C03642=1066.521,27.766,432.620,172.399,26.126,154.782
C03643=1066.516,27.517,432.635,172.398,26.123,154.782
C03644=1066.510,27.267,432.651,172.397,26.120,154.781
C03645=1066.504,27.017,432.666,172.395,26.118,154.781
C03646=1066.497,26.768,432.682,172.394,26.115,154.780
C03647=1066.492,26.518,432.698,172.392,26.112,154.780
C03648=1066.485,26.269,432.713,172.391,26.109,154.780
C03649=1066.480,26.020,432.728,172.389,26.107,154.780
C03650=1066.473,25.771,432.743,172.388,26.104,154.779
C03651=1066.467,25.521,432.760,172.386,26.102,154.779
C03652=1066.461,25.272,432.775,172.385,26.099,154.778
C03653=1066.455,25.022,432.790,172.384,26.096,154.778
C03654=1066.449,24.773,432.805,172.382,26.094,154.778
C03655=1066.444,24.523,432.821,172.381,26.091,154.777
C03656=1066.437,24.274,432.836,172.379,26.089,154.777
C03657=1066.431,24.024,432.852,172.378,26.086,154.777
C03658=1066.425,23.775,432.867,172.376,26.084,154.776
C03659=1066.420,23.525,432.882,172.375,26.081,154.776
C03660=1066.413,23.276,432.898,172.374,26.078,154.776
C03661=1066.408,23.026,432.913,172.372,26.075,154.775
C03662=1066.401,22.777,432.928,172.371,26.073,154.775
C03663=1066.396,22.527,432.944,172.369,26.070,154.775
C03664=1066.389,22.278,432.959,172.368,26.068,154.774
C03665=1066.384,22.028,432.975,172.366,26.065,154.774
C03666=1066.377,21.779,432.990,172.366,26.062,154.774
C03667=1066.372,21.529,433.005,172.365,26.060,154.773
C03668=1066.366,21.280,433.021,172.363,26.057,154.773
C03669=1066.360,21.030,433.036,172.362,26.055,154.773
C03670=1066.354,20.781,433.051,172.360,26.052,154.772
C03671=1066.348,20.532,433.066,172.359,26.050,154.772
C03672=1066.342,20.283,433.082,172.357,26.047,154.772
C03673=1066.336,20.033,433.097,172.356,26.045,154.771
C03674=1066.330,19.783,433.112,172.355,26.042,154.771
C03675=1066.324,19.534,433.127,172.353,26.039,154.771
C03676=1066.318,19.284,433.142,172.352,26.037,154.770
C03677=1066.312,19.034,433.157,172.350,26.034,154.770
C03678=1066.305,18.785,433.173,172.349,26.031,154.770
C03679=1066.300,18.536,433.188,172.347,26.029,154.769
C03680=1066.294,18.286,433.203,172.346,26.026,154.769
C03681=1066.288,18.037,433.218,172.344,26.024,154.769
C03682=1066.282,17.788,433.233,172.343,26.021,154.768
C03683=1066.276,17.538,433.248,172.342,26.019,154.768
C03684=1066.270,17.288,433.263,172.340,26.016,154.768
C03685=1066.264,17.040,433.279,172.339,26.013,154.767
C03686=1066.258,16.790,433.294,172.337,26.011,154.767
C03687=1066.252,16.540,433.309,172.336,26.008,154.767
C03688=1066.246,16.291,433.324,172.335,26.005,154.766
C03689=1066.240,16.041,433.339,172.333,26.003,154.766
C03690=1066.234,15.792,433.354,172.332,26.000,154.766
C03691=1066.228,15.543,433.369,172.330,25.998,154.765
C03692=1066.222,15.293,433.384,172.329,25.995,154.765
C03693=1066.216,15.043,433.399,172.327,25.993,154.765
C03694=1066.210,14.794,433.414,172.326,25.990,154.764
C03695=1066.203,14.511,433.431,172.324,25.987,154.764
C03696=1066.196,14.230,433.448,172.323,25.984,154.764
C03697=1066.189,13.948,433.465,172.322,25.982,154.763
C03698=1066.182,13.665,433.482,172.320,25.979,154.763
C03699=1066.176,13.416,433.497,172.319,25.976,154.763
C03700=1066.170,13.167,433.511,172.317,25.974,154.762
C03701=1066.164,12.917,433.527,172.316,25.971,154.762
C03702=1066.158,12.667,433.542,172.314,25.969,154.762
C03703=1066.152,12.418,433.556,172.313,25.966,154.761
C03704=1066.146,12.169,433.571,172.312,25.964,154.761
C03705=1066.140,11.919,433.586,172.310,25.961,154.761
C03706=1066.134,11.670,433.601,172.309,25.958,154.760
C03707=1066.128,11.420,433.615,172.307,25.956,154.760
C03708=1066.121,11.170,433.630,172.306,25.953,154.760
C03709=1066.115,10.921,433.644,172.304,25.951,154.759
C03710=1066.109,10.671,433.659,172.303,25.949,154.759
C03711=1066.103,10.422,433.674,172.302,25.946,154.759
C03712=1066.098,10.172,433.690,172.300,25.943,154.758
C03713=1066.091,9.923,433.704,172.299,25.941,154.758
C03714=1066.086,9.674,433.719,172.297,25.938,154.758
C03715=1066.079,9.424,433.734,172.296,25.936,154.757
C03716=1066.073,9.174,433.748,172.294,25.934,154.757
C03717=1066.067,8.925,433.763,172.293,25.931,154.757
C03718=1066.061,8.675,433.778,172.291,25.928,154.757
C03719=1066.055,8.426,433.792,172.290,25.925,154.756
C03720=1066.049,8.177,433.807,172.289,25.923,154.756
C03721=1066.042,7.927,433.822,172.287,25.921,154.756
C03722=1066.037,7.677,433.836,172.286,25.918,154.755
C03723=1066.030,7.428,433.851,172.284,25.916,154.755
C03724=1066.025,7.179,433.866,172.283,25.913,154.755
C03725=1066.018,6.929,433.881,172.281,25.910,154.754
C03726=1066.012,6.680,433.895,172.280,25.908,154.754
C03727=1066.006,6.430,433.909,172.278,25.906,154.754
C03728=1066.000,6.180,433.924,172.277,25.903,154.753
C03729=1065.994,5.931,433.939,172.276,25.901,154.753
C03730=1065.988,5.682,433.954,172.274,25.898,154.753
C03731=1065.982,5.432,433.968,172.273,25.895,154.752
C03732=1065.976,5.182,433.983,172.271,25.893,154.752
C03733=1065.970,4.934,433.997,172.270,25.890,154.752
C03734=1065.964,4.684,434.012,172.268,25.888,154.751
C03735=1065.958,4.434,434.026,172.267,25.885,154.751
C03736=1065.952,4.185,434.041,172.266,25.883,154.751
C03737=1065.946,3.936,434.056,172.265,25.881,154.751
C03738=1065.940,3.685,434.070,172.264,25.878,154.750
C03739=1065.934,3.436,434.084,172.262,25.875,154.750
C03740=1065.928,3.187,434.099,172.261,25.873,154.750
C03741=1065.923,2.937,434.113,172.259,25.871,154.749
C03742=1065.916,2.688,434.128,172.258,25.868,154.749
C03743=1065.910,2.439,434.143,172.256,25.865,154.749
C03744=1065.904,2.188,434.157,172.255,25.863,154.748
C03745=1065.898,1.939,434.172,172.254,25.860,154.748
C03746=1065.892,1.690,434.186,172.252,25.858,154.748
C03747=1065.887,1.440,434.200,172.251,25.856,154.747
C03748=1065.880,1.190,434.215,172.249,25.853,154.747
C03749=1065.875,0.941,434.229,172.248,25.850,154.747
C03750=1065.868,0.691,434.244,172.246,25.848,154.746
C03751=1065.863,0.442,434.259,172.245,25.845,154.746
C03752=1065.857,0.192,434.273,172.243,25.843,154.746
C03753=1065.851,-0.057,434.287,172.242,25.840,154.746
C03754=1065.845,-0.307,434.301,172.241,25.838,154.745
C03755=1065.839,-0.556,434.316,172.239,25.835,154.745
C03756=1065.833,-0.806,434.330,172.238,25.833,154.745
C03757=1065.827,-1.055,434.345,172.236,25.830,154.744
C03758=1065.822,-1.305,434.359,172.235,25.828,154.744
C03759=1065.815,-1.585,434.375,172.233,25.825,154.744
C03760=1065.808,-1.865,434.391,172.232,25.822,154.743
C03761=1065.801,-2.145,434.408,172.230,25.819,154.743
C03762=1065.794,-2.425,434.424,172.228,25.816,154.743
C03763=1065.788,-2.675,434.438,172.227,25.814,154.742
C03764=1065.783,-2.924,434.452,172.225,25.811,154.742
C03765=1065.777,-3.174,434.466,172.224,25.809,154.742
C03766=1065.771,-3.424,434.481,172.223,25.806,154.741
C03767=1065.765,-3.673,434.495,172.221,25.804,154.741
C03768=1065.758,-3.923,434.509,172.220,25.801,154.741
C03769=1065.753,-4.172,434.523,172.218,25.799,154.740
C03770=1065.747,-4.422,434.538,172.217,25.797,154.740
C03771=1065.740,-4.671,434.552,172.215,25.794,154.740
C03772=1065.734,-4.921,434.566,172.214,25.792,154.740
C03773=1065.728,-5.171,434.580,172.212,25.789,154.739
C03774=1065.722,-5.419,434.594,172.211,25.787,154.739
C03775=1065.716,-5.669,434.608,172.209,25.784,154.739
C03776=1065.710,-5.918,434.622,172.208,25.782,154.738
C03777=1065.704,-6.169,434.637,172.207,25.780,154.738
C03778=1065.698,-6.418,434.650,172.205,25.777,154.738
C03779=1065.691,-6.668,434.665,172.204,25.775,154.738
C03780=1065.686,-6.917,434.679,172.202,25.772,154.737
C03781=1065.680,-7.166,434.692,172.201,25.770,154.737
C03782=1065.673,-7.416,434.707,172.199,25.767,154.737
C03783=1065.667,-7.665,434.720,172.198,25.765,154.736
C03784=1065.661,-7.916,434.735,172.196,25.763,154.736
C03785=1065.655,-8.165,434.749,172.195,25.760,154.736
C03786=1065.649,-8.414,434.762,172.193,25.758,154.735
C03787=1065.643,-8.664,434.777,172.192,25.755,154.735
C03788=1065.637,-8.913,434.791,172.191,25.753,154.735
C03789=1065.631,-9.162,434.804,172.189,25.751,154.735
C03790=1065.625,-9.413,434.819,172.188,25.748,154.734
C03791=1065.619,-9.662,434.833,172.186,25.746,154.734
C03792=1065.613,-9.911,434.847,172.185,25.743,154.734
C03793=1065.607,-10.161,434.861,172.183,25.741,154.733
C03794=1065.601,-10.410,434.874,172.182,25.738,154.733
C03795=1065.595,-10.660,434.888,172.180,25.736,154.733
C03796=1065.589,-10.910,434.903,172.179,25.734,154.733
C03797=1065.583,-11.159,434.916,172.177,25.731,154.732
C03798=1065.577,-11.408,434.930,172.176,25.729,154.732
C03799=1065.571,-11.659,434.944,172.174,25.727,154.732
C03800=1065.565,-11.908,434.957,172.173,25.724,154.731
C03801=1065.559,-12.157,434.972,172.172,25.721,154.731
C03802=1065.552,-12.407,434.986,172.170,25.719,154.731
C03803=1065.547,-12.657,435.000,172.169,25.717,154.731
C03804=1065.541,-12.906,435.013,172.167,25.714,154.730
C03805=1065.535,-13.155,435.027,172.166,25.712,154.730
C03806=1065.529,-13.406,435.041,172.164,25.710,154.730
C03807=1065.522,-13.654,435.055,172.163,25.707,154.730
C03808=1065.517,-13.904,435.069,172.161,25.704,154.729
C03809=1065.511,-14.153,435.083,172.160,25.702,154.729
C03810=1065.505,-14.403,435.096,172.159,25.700,154.729
C03811=1065.499,-14.653,435.110,172.157,25.697,154.728
C03812=1065.493,-14.902,435.123,172.156,25.695,154.728
C03813=1065.487,-15.153,435.138,172.154,25.693,154.728
C03814=1065.481,-15.402,435.151,172.153,25.690,154.728
C03815=1065.475,-15.651,435.165,172.151,25.688,154.727
C03816=1065.469,-15.901,435.178,172.150,25.686,154.727
C03817=1065.462,-16.150,435.192,172.148,25.683,154.727
C03818=1065.456,-16.400,435.206,172.147,25.681,154.726
C03819=1065.450,-16.649,435.220,172.145,25.679,154.726
C03820=1065.444,-16.899,435.234,172.144,25.676,154.726
C03821=1065.438,-17.148,435.247,172.142,25.674,154.726
C03822=1065.432,-17.398,435.260,172.141,25.672,154.725
C03823=1065.425,-17.676,435.275,172.139,25.669,154.725
C03824=1065.418,-17.955,435.291,172.138,25.666,154.725
C03825=1065.411,-18.234,435.306,172.137,25.664,154.724
C03826=1065.405,-18.513,435.321,172.134,25.661,154.724
C03827=1065.398,-18.762,435.334,172.133,25.659,154.724
C03828=1065.393,-19.011,435.348,172.131,25.657,154.724
C03829=1065.387,-19.261,435.361,172.130,25.654,154.723
C03830=1065.380,-19.511,435.375,172.128,25.652,154.723
C03831=1065.374,-19.760,435.389,172.127,25.650,154.723
C03832=1065.368,-20.009,435.402,172.125,25.647,154.723
C03833=1065.363,-20.259,435.416,172.124,25.645,154.722
C03834=1065.356,-20.509,435.429,172.122,25.643,154.722
C03835=1065.350,-20.758,435.443,172.121,25.640,154.722
C03836=1065.344,-21.008,435.457,172.120,25.638,154.722
C03837=1065.338,-21.257,435.470,172.118,25.636,154.721
C03838=1065.332,-21.506,435.483,172.117,25.633,154.721
C03839=1065.326,-21.757,435.497,172.115,25.631,154.721
C03840=1065.320,-22.007,435.510,172.114,25.629,154.720
C03841=1065.314,-22.256,435.523,172.112,25.626,154.720
C03842=1065.308,-22.505,435.537,172.111,25.625,154.720
C03843=1065.302,-22.755,435.550,172.109,25.622,154.720
C03844=1065.296,-23.004,435.564,172.108,25.620,154.720
C03845=1065.290,-23.254,435.578,172.106,25.618,154.719
C03846=1065.284,-23.504,435.590,172.105,25.615,154.719
C03847=1065.277,-23.753,435.604,172.103,25.613,154.719
C03848=1065.271,-24.003,435.617,172.102,25.610,154.718
C03849=1065.266,-24.252,435.631,172.100,25.608,154.718
C03850=1065.260,-24.501,435.644,172.099,25.606,154.718
C03851=1065.253,-24.751,435.657,172.097,25.603,154.718
C03852=1065.248,-25.002,435.671,172.096,25.601,154.717
C03853=1065.241,-25.251,435.684,172.095,25.599,154.717
C03854=1065.235,-25.500,435.697,172.093,25.596,154.717
C03855=1065.230,-25.750,435.711,172.091,25.595,154.717
C03856=1065.224,-26.000,435.724,172.090,25.592,154.716
C03857=1065.218,-26.249,435.737,172.089,25.590,154.716
C03858=1065.211,-26.498,435.750,172.087,25.588,154.716
C03859=1065.206,-26.748,435.764,172.086,25.585,154.716
C03860=1065.200,-26.998,435.777,172.084,25.583,154.715
C03861=1065.193,-27.248,435.790,172.083,25.581,154.715
C03862=1065.187,-27.497,435.804,172.081,25.579,154.715
C03863=1065.181,-27.747,435.816,172.080,25.576,154.715
C03864=1065.175,-27.996,435.829,172.078,25.574,154.714
C03865=1065.169,-28.245,435.843,172.077,25.572,154.714
C03866=1065.162,-28.494,435.856,172.075,25.569,154.714
C03867=1065.156,-28.744,435.869,172.074,25.568,154.714
C03868=1065.151,-28.994,435.882,172.072,25.565,154.713
C03869=1065.144,-29.245,435.895,172.071,25.563,154.713
C03870=1065.138,-29.494,435.909,172.069,25.561,154.713
C03871=1065.132,-29.743,435.922,172.068,25.559,154.713
C03872=1065.126,-29.993,435.934,172.066,25.556,154.713
C03873=1065.120,-30.242,435.948,172.065,25.554,154.712
C03874=1065.114,-30.491,435.961,172.063,25.552,154.712
C03875=1065.108,-30.741,435.974,172.062,25.550,154.712
C03876=1065.102,-30.991,435.987,172.060,25.548,154.712
C03877=1065.096,-31.240,435.999,172.059,25.545,154.711
C03878=1065.089,-31.490,436.013,172.057,25.543,154.711
C03879=1065.083,-31.739,436.026,172.056,25.541,154.711
C03880=1065.077,-31.989,436.038,172.054,25.539,154.711
C03881=1065.071,-32.239,436.052,172.053,25.537,154.710
C03882=1065.065,-32.489,436.065,172.051,25.534,154.710
C03883=1065.058,-32.738,436.078,172.050,25.532,154.710
C03884=1065.052,-32.988,436.090,172.048,25.530,154.710
C03885=1065.046,-33.237,436.104,172.047,25.528,154.709
C03886=1065.040,-33.487,436.116,172.045,25.526,154.709
C03887=1065.034,-33.765,436.131,172.043,25.523,154.709
C03888=1065.027,-34.042,436.146,172.041,25.521,154.709
C03889=1065.020,-34.320,436.160,172.040,25.519,154.709
C03890=1065.014,-34.598,436.175,172.038,25.516,154.708
C03891=1065.008,-34.848,436.187,172.037,25.514,154.708
C03892=1065.002,-35.097,436.201,172.036,25.511,154.708
C03893=1064.996,-35.347,436.213,172.034,25.509,154.707
C03894=1064.990,-35.596,436.226,172.033,25.507,154.707
C03895=1064.984,-35.846,436.239,172.031,25.505,154.707
C03896=1064.978,-36.096,436.252,172.029,25.502,154.707
C03897=1064.972,-36.345,436.265,172.027,25.501,154.707
C03898=1064.966,-36.595,436.277,172.026,25.498,154.706
C03899=1064.959,-36.844,436.291,172.024,25.496,154.706
C03900=1064.954,-37.094,436.303,172.023,25.494,154.706
C03901=1064.947,-37.344,436.317,172.021,25.492,154.706
C03902=1064.941,-37.593,436.329,172.020,25.489,154.705
C03903=1064.936,-37.843,436.342,172.018,25.488,154.705
C03904=1064.930,-38.092,436.355,172.017,25.485,154.705
C03905=1064.924,-38.342,436.367,172.015,25.483,154.705
C03906=1064.918,-38.592,436.380,172.014,25.481,154.705
C03907=1064.911,-38.841,436.392,172.012,25.479,154.704
C03908=1064.905,-39.090,436.405,172.011,25.477,154.704
C03909=1064.899,-39.340,436.418,172.009,25.475,154.704
C03910=1064.893,-39.590,436.431,172.008,25.472,154.704
C03911=1064.887,-39.839,436.443,172.006,25.471,154.704
C03912=1064.881,-40.089,436.455,172.005,25.468,154.703
C03913=1064.874,-40.338,436.468,172.003,25.466,154.703
C03914=1064.868,-40.588,436.481,172.002,25.464,154.703
C03915=1064.863,-40.838,436.494,172.000,25.462,154.703
C03916=1064.856,-41.087,436.506,171.999,25.460,154.702
C03917=1064.850,-41.337,436.519,171.997,25.458,154.702
C03918=1064.844,-41.587,436.531,171.995,25.456,154.702
C03919=1064.838,-41.837,436.544,171.994,25.454,154.702
C03920=1064.832,-42.086,436.557,171.992,25.452,154.702
C03921=1064.825,-42.336,436.569,171.991,25.450,154.701
C03922=1064.819,-42.585,436.582,171.989,25.447,154.701
C03923=1064.813,-42.835,436.594,171.988,25.446,154.701
C03924=1064.807,-43.085,436.608,171.986,25.443,154.701
C03925=1064.801,-43.333,436.619,171.985,25.442,154.701
C03926=1064.795,-43.583,436.632,171.983,25.439,154.700
C03927=1064.789,-43.833,436.644,171.982,25.437,154.700
C03928=1064.783,-44.083,436.657,171.980,25.435,154.700
C03929=1064.776,-44.332,436.669,171.978,25.433,154.700
C03930=1064.770,-44.582,436.682,171.976,25.431,154.700
C03931=1064.764,-44.832,436.695,171.975,25.429,154.699
C03932=1064.759,-45.082,436.707,171.973,25.426,154.699
C03933=1064.752,-45.331,436.719,171.972,25.425,154.699
C03934=1064.747,-45.580,436.731,171.970,25.423,154.699
C03935=1064.740,-45.830,436.745,171.969,25.421,154.699
C03936=1064.734,-46.080,436.757,171.967,25.419,154.699
C03937=1064.728,-46.329,436.769,171.966,25.416,154.698
C03938=1064.722,-46.579,436.782,171.964,25.415,154.698
C03939=1064.716,-46.829,436.794,171.963,25.412,154.698
C03940=1064.709,-47.078,436.806,171.961,25.411,154.698
C03941=1064.704,-47.328,436.818,171.960,25.408,154.697
C03942=1064.698,-47.578,436.831,171.958,25.406,154.697
C03943=1064.692,-47.827,436.843,171.956,25.405,154.697
C03944=1064.685,-48.076,436.856,171.955,25.402,154.697
C03945=1064.679,-48.326,436.869,171.953,25.400,154.697
C03946=1064.674,-48.575,436.881,171.952,25.398,154.696
C03947=1064.667,-48.825,436.893,171.950,25.396,154.696
C03948=1064.661,-49.075,436.905,171.949,25.394,154.696
C03949=1064.656,-49.325,436.918,171.947,25.392,154.696
C03950=1064.649,-49.574,436.930,171.946,25.390,154.696
C03951=1064.642,-49.853,436.943,171.943,25.388,154.696
C03952=1064.636,-50.131,436.957,171.942,25.385,154.695
C03953=1064.629,-50.409,436.971,171.940,25.384,154.695
C03954=1064.622,-50.687,436.984,171.939,25.381,154.695
C03955=1064.616,-50.937,436.997,171.937,25.379,154.695
C03956=1064.610,-51.187,437.009,171.936,25.378,154.695
C03957=1064.604,-51.435,437.020,171.934,25.376,154.694
C03958=1064.598,-51.685,437.033,171.933,25.373,154.694
C03959=1064.591,-51.935,437.045,171.930,25.371,154.694
C03960=1064.585,-52.185,437.058,171.929,25.370,154.694
C03961=1064.578,-52.434,437.069,171.927,25.368,154.694
C03962=1064.572,-52.684,437.081,171.925,25.366,154.694
C03963=1064.567,-52.934,437.093,171.924,25.364,154.693
C03964=1064.560,-53.183,437.105,171.922,25.362,154.693
C03965=1064.554,-53.433,437.117,171.921,25.360,154.693
C03966=1064.548,-53.683,437.129,171.919,25.358,154.693
C03967=1064.541,-53.932,437.141,171.918,25.357,154.693
C03968=1064.535,-54.182,437.154,171.916,25.355,154.693
C03969=1064.529,-54.431,437.165,171.915,25.352,154.692
C03970=1064.523,-54.681,437.178,171.913,25.351,154.692
C03971=1064.516,-54.930,437.190,171.911,25.349,154.692
C03972=1064.510,-55.181,437.201,171.910,25.347,154.692
C03973=1064.505,-55.430,437.213,171.908,25.345,154.692
C03974=1064.498,-55.679,437.225,171.907,25.343,154.692
C03975=1064.492,-55.929,437.237,171.905,25.342,154.692
C03976=1064.486,-56.179,437.250,171.904,25.339,154.691
C03977=1064.479,-56.429,437.261,171.902,25.337,154.691
C03978=1064.473,-56.678,437.273,171.900,25.336,154.691
C03979=1064.467,-56.928,437.285,171.899,25.334,154.691
C03980=1064.461,-57.177,437.297,171.897,25.332,154.691
C03981=1064.454,-57.427,437.309,171.895,25.330,154.691
C03982=1064.449,-57.677,437.321,171.893,25.328,154.690
C03983=1064.442,-57.926,437.333,171.892,25.326,154.690
C03984=1064.436,-58.176,437.345,171.890,25.324,154.690
C03985=1064.430,-58.425,437.357,171.889,25.322,154.690
C03986=1064.424,-58.675,437.368,171.887,25.321,154.690
C03987=1064.418,-58.925,437.381,171.885,25.319,154.690
C03988=1064.412,-59.175,437.393,171.884,25.317,154.690
C03989=1064.405,-59.424,437.404,171.882,25.315,154.689
C03990=1064.399,-59.674,437.415,171.881,25.313,154.689
C03991=1064.393,-59.924,437.428,171.879,25.312,154.689
C03992=1064.387,-60.173,437.440,171.878,25.310,154.689
C03993=1064.381,-60.423,437.451,171.876,25.308,154.689
C03994=1064.375,-60.673,437.463,171.874,25.306,154.689
C03995=1064.369,-60.922,437.475,171.873,25.304,154.689
C03996=1064.363,-61.172,437.486,171.871,25.303,154.688
C03997=1064.357,-61.422,437.499,171.870,25.300,154.688
C03998=1064.351,-61.670,437.510,171.868,25.298,154.688
C03999=1064.344,-61.921,437.522,171.867,25.297,154.688
C04000=1064.338,-62.171,437.534,171.865,25.295,154.688
C04001=1064.332,-62.419,437.546,171.864,25.293,154.688
C04002=1064.326,-62.670,437.557,171.862,25.291,154.687
C04003=1064.319,-62.919,437.569,171.859,25.289,154.687
C04004=1064.314,-63.169,437.580,171.858,25.287,154.687
C04005=1064.308,-63.419,437.592,171.856,25.286,154.687
C04006=1064.301,-63.668,437.604,171.855,25.284,154.687
C04007=1064.296,-63.918,437.616,171.853,25.282,154.687
C04008=1064.289,-64.167,437.628,171.852,25.280,154.687
C04009=1064.284,-64.417,437.639,171.850,25.278,154.686
C04010=1064.277,-64.667,437.651,171.848,25.277,154.686
C04011=1064.271,-64.917,437.662,171.847,25.275,154.686
C04012=1064.265,-65.166,437.674,171.845,25.273,154.686
C04013=1064.259,-65.416,437.685,171.844,25.271,154.686
C04014=1064.253,-65.665,437.697,171.842,25.270,154.686
C04015=1064.246,-65.945,437.710,171.841,25.268,154.686
C04016=1064.239,-66.224,437.723,171.838,25.266,154.686
C04017=1064.232,-66.504,437.736,171.836,25.264,154.685
C04018=1064.226,-66.783,437.749,171.835,25.261,154.685
C04019=1064.220,-67.033,437.761,171.833,25.260,154.685
C04020=1064.214,-67.282,437.772,171.832,25.258,154.685
C04021=1064.208,-67.533,437.784,171.830,25.257,154.685
C04022=1064.201,-67.782,437.796,171.829,25.255,154.685
C04023=1064.196,-68.032,437.806,171.827,25.253,154.685
C04024=1064.190,-68.282,437.819,171.825,25.251,154.684
C04025=1064.184,-68.531,437.830,171.824,25.249,154.684
C04026=1064.177,-68.781,437.842,171.821,25.247,154.684
C04027=1064.172,-69.030,437.853,171.820,25.246,154.684
C04028=1064.166,-69.280,437.865,171.818,25.244,154.684
C04029=1064.160,-69.529,437.876,171.817,25.242,154.684
C04030=1064.154,-69.780,437.887,171.815,25.240,154.684
C04031=1064.148,-70.028,437.899,171.813,25.238,154.683
C04032=1064.141,-70.279,437.910,171.812,25.237,154.683
C04033=1064.136,-70.528,437.922,171.810,25.235,154.683
C04034=1064.130,-70.778,437.934,171.809,25.234,154.683
C04035=1064.124,-71.028,437.944,171.807,25.232,154.683
C04036=1064.117,-71.277,437.956,171.805,25.230,154.683
C04037=1064.111,-71.527,437.967,171.804,25.228,154.683
C04038=1064.106,-71.777,437.979,171.802,25.226,154.683
C04039=1064.100,-72.026,437.991,171.801,25.225,154.682
C04040=1064.094,-72.275,438.002,171.799,25.223,154.682
C04041=1064.088,-72.526,438.013,171.797,25.222,154.682
C04042=1064.082,-72.775,438.024,171.796,25.220,154.682
C04043=1064.076,-73.025,438.036,171.794,25.218,154.682
C04044=1064.070,-73.275,438.047,171.793,25.216,154.682
C04045=1064.064,-73.524,438.059,171.791,25.214,154.682
C04046=1064.058,-73.774,438.070,171.790,25.213,154.682
C04047=1064.052,-74.024,438.081,171.787,25.211,154.682
C04048=1064.046,-74.273,438.092,171.785,25.209,154.681
C04049=1064.039,-74.523,438.104,171.784,25.208,154.681
C04050=1064.033,-74.772,438.115,171.782,25.206,154.681
C04051=1064.027,-75.023,438.126,171.780,25.204,154.681
C04052=1064.021,-75.272,438.137,171.779,25.203,154.681
C04053=1064.015,-75.521,438.149,171.777,25.201,154.681
C04054=1064.009,-75.771,438.160,171.776,25.200,154.681
C04055=1064.003,-76.021,438.171,171.774,25.198,154.681
C04056=1063.997,-76.271,438.182,171.772,25.196,154.681
C04057=1063.991,-76.520,438.193,171.771,25.195,154.681
C04058=1063.985,-76.770,438.205,171.769,25.193,154.680
C04059=1063.979,-77.019,438.216,171.768,25.191,154.680
C04060=1063.972,-77.270,438.227,171.766,25.190,154.680
C04061=1063.967,-77.519,438.238,171.764,25.188,154.680
C04062=1063.960,-77.769,438.249,171.763,25.187,154.680
C04063=1063.954,-78.018,438.259,171.761,25.185,154.680
C04064=1063.948,-78.268,438.270,171.759,25.183,154.680
C04065=1063.942,-78.517,438.282,171.758,25.182,154.680
C04066=1063.936,-78.767,438.293,171.756,25.180,154.680
C04067=1063.929,-79.017,438.304,171.755,25.179,154.680
C04068=1063.924,-79.267,438.315,171.752,25.177,154.680
C04069=1063.918,-79.516,438.326,171.750,25.175,154.679
C04070=1063.912,-79.766,438.337,171.749,25.174,154.679
C04071=1063.906,-80.016,438.348,171.747,25.172,154.679
C04072=1063.899,-80.266,438.359,171.745,25.171,154.679
C04073=1063.893,-80.515,438.370,171.744,25.169,154.679
C04074=1063.887,-80.765,438.381,171.742,25.168,154.679
C04075=1063.881,-81.014,438.393,171.741,25.166,154.679
C04076=1063.874,-81.263,438.403,171.739,25.165,154.679
C04077=1063.868,-81.514,438.414,171.737,25.163,154.679
C04078=1063.862,-81.763,438.425,171.736,25.162,154.679
C04079=1063.855,-82.045,438.437,171.734,25.160,154.679
C04080=1063.848,-82.327,438.449,171.731,25.159,154.679
C04081=1063.841,-82.609,438.461,171.730,25.157,154.678
C04082=1063.834,-82.890,438.474,171.728,25.156,154.678
C04083=1063.828,-83.140,438.484,171.727,25.154,154.678
C04084=1063.821,-83.390,438.495,171.725,25.153,154.678
C04085=1063.815,-83.639,438.506,171.723,25.151,154.678
C04086=1063.810,-83.889,438.517,171.722,25.150,154.678
C04087=1063.803,-84.139,438.527,171.719,25.148,154.678
C04088=1063.797,-84.388,438.538,171.717,25.146,154.678
C04089=1063.791,-84.638,438.550,171.716,25.145,154.678
C04090=1063.784,-84.887,438.560,171.714,25.143,154.678
C04091=1063.778,-85.137,438.571,171.712,25.142,154.678
C04092=1063.772,-85.387,438.582,171.711,25.141,154.678
C04093=1063.766,-85.637,438.593,171.709,25.139,154.678
C04094=1063.760,-85.886,438.603,171.707,25.138,154.678
C04095=1063.753,-86.136,438.614,171.706,25.137,154.678
C04096=1063.748,-86.385,438.625,171.704,25.135,154.678
C04097=1063.741,-86.635,438.635,171.702,25.134,154.678
C04098=1063.735,-86.885,438.646,171.701,25.132,154.678
C04099=1063.729,-87.135,438.657,171.699,25.131,154.677
C04100=1063.723,-87.384,438.667,171.697,25.129,154.677
C04101=1063.717,-87.634,438.678,171.696,25.128,154.677
C04102=1063.711,-87.884,438.689,171.694,25.126,154.677
C04103=1063.704,-88.133,438.700,171.692,25.125,154.677
C04104=1063.698,-88.384,438.710,171.691,25.124,154.677
C04105=1063.692,-88.633,438.720,171.689,25.123,154.677
C04106=1063.686,-88.882,438.731,171.687,25.121,154.677
C04107=1063.680,-89.132,438.742,171.686,25.120,154.677
C04108=1063.673,-89.382,438.753,171.683,25.118,154.677
C04109=1063.668,-89.632,438.763,171.681,25.116,154.677
C04110=1063.662,-89.881,438.774,171.680,25.115,154.677
C04111=1063.655,-90.131,438.785,171.678,25.114,154.677
C04112=1063.649,-90.381,438.795,171.676,25.113,154.677
C04113=1063.644,-90.630,438.806,171.675,25.111,154.677
C04114=1063.637,-90.880,438.816,171.673,25.110,154.677
C04115=1063.631,-91.130,438.827,171.671,25.108,154.677
C04116=1063.625,-91.379,438.837,171.670,25.107,154.677
C04117=1063.619,-91.629,438.848,171.668,25.105,154.676
C04118=1063.613,-91.879,438.858,171.666,25.104,154.676
C04119=1063.607,-92.128,438.869,171.665,25.103,154.676
C04120=1063.601,-92.378,438.880,171.663,25.102,154.676
C04121=1063.594,-92.628,438.890,171.661,25.100,154.676
C04122=1063.589,-92.878,438.900,171.660,25.099,154.676
C04123=1063.583,-93.127,438.911,171.658,25.097,154.676
C04124=1063.576,-93.377,438.922,171.656,25.096,154.676
C04125=1063.570,-93.627,438.932,171.655,25.095,154.676
C04126=1063.564,-93.876,438.942,171.653,25.094,154.676
C04127=1063.558,-94.126,438.953,171.651,25.092,154.676
C04128=1063.553,-94.376,438.963,171.650,25.091,154.676
C04129=1063.546,-94.625,438.974,171.648,25.090,154.676
C04130=1063.540,-94.876,438.984,171.646,25.088,154.676
C04131=1063.534,-95.125,438.994,171.644,25.087,154.676
C04132=1063.528,-95.375,439.005,171.642,25.086,154.676
C04133=1063.522,-95.624,439.015,171.640,25.084,154.676
C04134=1063.516,-95.874,439.026,171.639,25.082,154.676
C04135=1063.510,-96.123,439.037,171.637,25.081,154.676
C04136=1063.504,-96.374,439.047,171.635,25.080,154.676
C04137=1063.498,-96.623,439.057,171.633,25.079,154.676
C04138=1063.492,-96.873,439.067,171.632,25.078,154.676
C04139=1063.486,-97.123,439.078,171.630,25.076,154.676
C04140=1063.480,-97.372,439.088,171.628,25.075,154.676
C04141=1063.474,-97.622,439.098,171.627,25.073,154.676
C04142=1063.467,-97.872,439.109,171.625,25.072,154.676
C04143=1063.461,-98.156,439.121,171.623,25.071,154.676
C04144=1063.453,-98.440,439.132,171.621,25.069,154.676
C04145=1063.447,-98.724,439.143,171.619,25.068,154.676
C04146=1063.440,-99.008,439.156,171.617,25.067,154.676
C04147=1063.433,-99.258,439.165,171.616,25.066,154.676
C04148=1063.427,-99.507,439.175,171.614,25.064,154.676
C04149=1063.421,-99.757,439.186,171.612,25.063,154.676
C04150=1063.415,-100.006,439.196,171.610,25.062,154.676
C04151=1063.408,-100.257,439.206,171.609,25.061,154.676
C04152=1063.402,-100.506,439.217,171.607,25.060,154.676
C04153=1063.396,-100.756,439.226,171.604,25.059,154.676
C04154=1063.390,-101.005,439.237,171.603,25.057,154.676
C04155=1063.384,-101.255,439.247,171.601,25.056,154.676
C04156=1063.378,-101.505,439.256,171.599,25.055,154.676
C04157=1063.372,-101.754,439.267,171.597,25.054,154.676
C04158=1063.366,-102.004,439.277,171.596,25.052,154.676
C04159=1063.359,-102.254,439.287,171.594,25.051,154.676
C04160=1063.353,-102.504,439.297,171.592,25.050,154.676
C04161=1063.347,-102.753,439.308,171.590,25.049,154.676
C04162=1063.341,-103.003,439.317,171.589,25.048,154.676
C04163=1063.335,-103.253,439.327,171.587,25.047,154.676
C04164=1063.329,-103.502,439.338,171.585,25.046,154.676
C04165=1063.323,-103.752,439.347,171.584,25.044,154.676
C04166=1063.317,-104.002,439.357,171.582,25.043,154.676
C04167=1063.310,-104.251,439.367,171.580,25.042,154.676
C04168=1063.305,-104.501,439.377,171.578,25.041,154.676
C04169=1063.298,-104.750,439.388,171.577,25.040,154.676
C04170=1063.292,-105.001,439.398,171.575,25.039,154.676
C04171=1063.286,-105.251,439.408,171.573,25.038,154.676
C04172=1063.280,-105.500,439.418,171.572,25.036,154.676
C04173=1063.274,-105.750,439.428,171.570,25.036,154.676
C04174=1063.267,-106.000,439.437,171.568,25.035,154.676
C04175=1063.262,-106.250,439.447,171.566,25.033,154.676
C04176=1063.256,-106.499,439.458,171.565,25.032,154.676
C04177=1063.249,-106.749,439.467,171.563,25.032,154.676
C04178=1063.243,-106.999,439.477,171.561,25.030,154.676
C04179=1063.237,-107.248,439.488,171.559,25.029,154.676
C04180=1063.231,-107.498,439.497,171.558,25.028,154.676
C04181=1063.225,-107.748,439.507,171.555,25.027,154.676
C04182=1063.219,-107.998,439.516,171.553,25.026,154.676
C04183=1063.212,-108.247,439.527,171.551,25.024,154.676
C04184=1063.206,-108.497,439.536,171.550,25.024,154.676
C04185=1063.200,-108.746,439.546,171.548,25.023,154.676
C04186=1063.195,-108.997,439.556,171.546,25.021,154.676
C04187=1063.188,-109.246,439.565,171.544,25.021,154.676
C04188=1063.182,-109.495,439.576,171.543,25.019,154.676
C04189=1063.176,-109.745,439.585,171.541,25.019,154.676
C04190=1063.170,-109.995,439.595,171.539,25.018,154.676
C04191=1063.164,-110.245,439.604,171.537,25.016,154.676
C04192=1063.157,-110.495,439.614,171.536,25.016,154.676
C04193=1063.151,-110.744,439.624,171.534,25.015,154.676
C04194=1063.145,-110.994,439.634,171.532,25.014,154.676
C04195=1063.139,-111.244,439.644,171.530,25.013,154.676
C04196=1063.133,-111.494,439.654,171.529,25.011,154.676
C04197=1063.127,-111.743,439.663,171.527,25.011,154.676
C04198=1063.121,-111.993,439.673,171.525,25.010,154.676
C04199=1063.115,-112.243,439.682,171.523,25.009,154.676
C04200=1063.108,-112.493,439.692,171.522,25.008,154.676
C04201=1063.102,-112.742,439.702,171.520,25.007,154.677
C04202=1063.096,-112.992,439.712,171.518,25.006,154.677
C04203=1063.090,-113.242,439.721,171.516,25.005,154.677
C04204=1063.083,-113.491,439.731,171.514,25.004,154.677
C04205=1063.077,-113.741,439.740,171.513,25.003,154.677
C04206=1063.071,-113.991,439.750,171.511,25.002,154.677
C04207=1063.064,-114.273,439.761,171.508,25.001,154.677
C04208=1063.057,-114.555,439.772,171.506,25.000,154.677
C04209=1063.051,-114.838,439.783,171.505,24.999,154.677
C04210=1063.044,-115.120,439.793,171.503,24.998,154.677
C04211=1063.037,-115.370,439.803,171.501,24.997,154.677
C04212=1063.031,-115.620,439.812,171.499,24.996,154.677
C04213=1063.025,-115.869,439.822,171.497,24.995,154.677
C04214=1063.019,-116.119,439.832,171.496,24.994,154.677
C04215=1063.013,-116.369,439.841,171.493,24.993,154.677
C04216=1063.007,-116.619,439.851,171.491,24.992,154.677
C04217=1063.001,-116.868,439.860,171.489,24.991,154.677
C04218=1062.995,-117.118,439.870,171.488,24.990,154.677
C04219=1062.989,-117.368,439.879,171.486,24.990,154.677
C04220=1062.982,-117.617,439.889,171.484,24.989,154.678
C04221=1062.976,-117.867,439.898,171.482,24.988,154.678
C04222=1062.970,-118.117,439.908,171.480,24.987,154.678
C04223=1062.964,-118.367,439.917,171.479,24.986,154.678
C04224=1062.957,-118.616,439.926,171.477,24.985,154.678
C04225=1062.951,-118.866,439.936,171.475,24.985,154.678
C04226=1062.945,-119.116,439.945,171.473,24.984,154.678
C04227=1062.939,-119.365,439.955,171.472,24.983,154.678
C04228=1062.933,-119.615,439.964,171.470,24.982,154.678
C04229=1062.927,-119.864,439.974,171.468,24.981,154.678
C04230=1062.921,-120.115,439.983,171.466,24.980,154.678
C04231=1062.915,-120.365,439.992,171.464,24.979,154.678
C04232=1062.909,-120.614,440.002,171.462,24.979,154.678
C04233=1062.902,-120.864,440.011,171.461,24.978,154.678
C04234=1062.895,-121.114,440.020,171.459,24.977,154.678
C04235=1062.890,-121.363,440.030,171.457,24.976,154.679
C04236=1062.884,-121.613,440.039,171.455,24.976,154.679
C04237=1062.878,-121.863,440.048,171.453,24.975,154.679
C04238=1062.872,-122.113,440.058,171.452,24.974,154.679
C04239=1062.866,-122.363,440.067,171.450,24.973,154.679
C04240=1062.859,-122.612,440.077,171.448,24.973,154.679
C04241=1062.852,-122.862,440.086,171.446,24.972,154.679
C04242=1062.847,-123.112,440.094,171.444,24.971,154.679
C04243=1062.841,-123.361,440.104,171.443,24.970,154.679
C04244=1062.835,-123.611,440.113,171.441,24.969,154.679
C04245=1062.829,-123.861,440.123,171.439,24.969,154.679
C04246=1062.823,-124.111,440.132,171.437,24.968,154.679
C04247=1062.817,-124.360,440.140,171.435,24.967,154.679
C04248=1062.810,-124.610,440.150,171.433,24.966,154.680
C04249=1062.804,-124.860,440.159,171.432,24.966,154.680
C04250=1062.798,-125.110,440.169,171.430,24.965,154.680
C04251=1062.791,-125.360,440.177,171.428,24.964,154.680
C04252=1062.785,-125.610,440.187,171.426,24.964,154.680
C04253=1062.780,-125.859,440.196,171.424,24.963,154.680
C04254=1062.773,-126.108,440.206,171.422,24.962,154.680
C04255=1062.767,-126.359,440.214,171.421,24.962,154.680
C04256=1062.761,-126.608,440.223,171.419,24.961,154.680
C04257=1062.755,-126.858,440.233,171.417,24.960,154.681
C04258=1062.749,-127.108,440.241,171.415,24.959,154.681
C04259=1062.742,-127.357,440.250,171.413,24.959,154.681
C04260=1062.736,-127.607,440.260,171.411,24.958,154.681
C04261=1062.730,-127.858,440.269,171.410,24.957,154.681
C04262=1062.725,-128.107,440.279,171.408,24.956,154.681
C04263=1062.722,-128.357,440.288,171.406,24.954,154.681
C04264=1062.720,-128.609,440.300,171.405,24.952,154.680
C04265=1062.720,-128.859,440.312,171.404,24.949,154.680
C04266=1062.720,-129.109,440.325,171.403,24.945,154.680
C04267=1062.723,-129.362,440.338,171.402,24.941,154.679
C04268=1062.727,-129.613,440.352,171.402,24.937,154.678
C04269=1062.733,-129.864,440.367,171.401,24.931,154.677
C04270=1062.741,-130.115,440.383,171.400,24.925,154.676
C04271=1062.358,-130.137,440.196,171.353,25.079,154.709
C04272=1062.351,-129.887,440.180,171.354,25.085,154.710
C04273=1062.346,-129.636,440.165,171.354,25.090,154.711
C04274=1062.341,-129.384,440.150,171.354,25.095,154.712
C04275=1062.339,-129.132,440.138,171.355,25.100,154.713
C04276=1062.338,-128.881,440.124,171.356,25.103,154.713
C04277=1062.338,-128.631,440.113,171.358,25.106,154.713
C04278=1062.340,-128.381,440.101,171.359,25.109,154.714
C04279=1062.344,-128.130,440.091,171.360,25.110,154.714
C04280=1062.347,-127.879,440.081,171.361,25.111,154.714
C04281=1062.354,-127.630,440.072,171.363,25.112,154.714
C04282=1062.360,-127.381,440.063,171.365,25.113,154.714
C04283=1062.366,-127.131,440.053,171.367,25.113,154.714
C04284=1062.373,-126.881,440.045,171.369,25.114,154.714
C04285=1062.379,-126.631,440.036,171.371,25.114,154.713
C04286=1062.385,-126.381,440.026,171.373,25.115,154.713
C04287=1062.390,-126.131,440.017,171.375,25.116,154.713
C04288=1062.397,-125.882,440.008,171.377,25.117,154.713
C04289=1062.403,-125.632,439.999,171.379,25.118,154.713
C04290=1062.409,-125.382,439.990,171.381,25.119,154.713
C04291=1062.415,-125.132,439.981,171.383,25.119,154.713
C04292=1062.422,-124.883,439.972,171.384,25.120,154.713
C04293=1062.428,-124.633,439.962,171.386,25.120,154.713
C04294=1062.434,-124.383,439.953,171.388,25.121,154.713
C04295=1062.440,-124.133,439.944,171.390,25.122,154.712
C04296=1062.447,-123.884,439.935,171.392,25.122,154.712
C04297=1062.453,-123.634,439.925,171.394,25.124,154.712
C04298=1062.458,-123.385,439.916,171.395,25.124,154.712
C04299=1062.464,-123.134,439.907,171.397,25.125,154.712
C04300=1062.470,-122.884,439.898,171.399,25.125,154.712
C04301=1062.477,-122.635,439.888,171.401,25.126,154.712
C04302=1062.484,-122.385,439.879,171.403,25.127,154.712
C04303=1062.490,-122.135,439.870,171.404,25.128,154.712
C04304=1062.495,-121.886,439.861,171.406,25.129,154.712
C04305=1062.501,-121.636,439.852,171.408,25.129,154.712
C04306=1062.507,-121.386,439.842,171.410,25.130,154.712
C04307=1062.514,-121.136,439.832,171.412,25.131,154.712
C04308=1062.520,-120.886,439.823,171.414,25.132,154.711
C04309=1062.527,-120.637,439.814,171.415,25.132,154.711
C04310=1062.533,-120.387,439.804,171.417,25.134,154.711
C04311=1062.538,-120.138,439.796,171.419,25.134,154.711
C04312=1062.544,-119.888,439.786,171.421,25.135,154.711
C04313=1062.550,-119.638,439.777,171.423,25.135,154.711
C04314=1062.557,-119.388,439.767,171.424,25.137,154.711
C04315=1062.563,-119.138,439.758,171.426,25.137,154.711
C04316=1062.569,-118.889,439.748,171.428,25.138,154.711
C04317=1062.575,-118.639,439.738,171.430,25.139,154.711
C04318=1062.581,-118.389,439.729,171.432,25.140,154.711
C04319=1062.587,-118.139,439.719,171.434,25.140,154.711
C04320=1062.594,-117.890,439.711,171.435,25.142,154.711
C04321=1062.600,-117.641,439.701,171.437,25.142,154.711
C04322=1062.606,-117.391,439.692,171.439,25.143,154.710
C04323=1062.612,-117.141,439.682,171.441,25.144,154.710
C04324=1062.618,-116.891,439.672,171.442,25.145,154.710
C04325=1062.625,-116.641,439.663,171.444,25.146,154.710
C04326=1062.631,-116.392,439.653,171.446,25.147,154.710
C04327=1062.637,-116.142,439.644,171.448,25.147,154.710
C04328=1062.643,-115.892,439.634,171.450,25.148,154.710
C04329=1062.649,-115.642,439.625,171.451,25.149,154.710
C04330=1062.655,-115.392,439.615,171.453,25.150,154.710
C04331=1062.662,-115.143,439.605,171.455,25.151,154.710
C04332=1062.669,-114.860,439.595,171.458,25.153,154.710
C04333=1062.675,-114.578,439.584,171.460,25.153,154.710
C04334=1062.683,-114.296,439.573,171.461,25.154,154.710
C04335=1062.689,-114.013,439.562,171.464,25.155,154.710
C04336=1062.695,-113.764,439.553,171.466,25.157,154.710
C04337=1062.701,-113.514,439.543,171.468,25.157,154.710
C04338=1062.708,-113.264,439.533,171.469,25.158,154.710
C04339=1062.714,-113.014,439.524,171.471,25.159,154.709
C04340=1062.720,-112.764,439.514,171.473,25.160,154.709
C04341=1062.726,-112.515,439.505,171.475,25.161,154.709
C04342=1062.732,-112.265,439.495,171.476,25.162,154.709
C04343=1062.738,-112.015,439.486,171.478,25.163,154.709
C04344=1062.744,-111.766,439.475,171.480,25.164,154.709
C04345=1062.750,-111.516,439.466,171.482,25.165,154.709
C04346=1062.756,-111.267,439.456,171.484,25.166,154.709
C04347=1062.762,-111.017,439.446,171.485,25.167,154.709
C04348=1062.768,-110.767,439.437,171.487,25.168,154.709
C04349=1062.774,-110.517,439.427,171.489,25.169,154.709
C04350=1062.781,-110.267,439.418,171.490,25.170,154.709
C04351=1062.787,-110.018,439.407,171.492,25.171,154.709
C04352=1062.794,-109.768,439.397,171.494,25.172,154.709
C04353=1062.800,-109.518,439.388,171.496,25.173,154.709
C04354=1062.805,-109.268,439.378,171.498,25.174,154.709
C04355=1062.812,-109.018,439.368,171.499,25.175,154.709
C04356=1062.818,-108.769,439.358,171.501,25.176,154.709
C04357=1062.824,-108.519,439.348,171.503,25.177,154.709
C04358=1062.830,-108.269,439.339,171.505,25.178,154.709
C04359=1062.837,-108.020,439.329,171.506,25.179,154.709
C04360=1062.843,-107.770,439.319,171.508,25.180,154.709
C04361=1062.849,-107.521,439.309,171.511,25.181,154.709
C04362=1062.855,-107.270,439.299,171.513,25.182,154.709
C04363=1062.861,-107.021,439.290,171.514,25.183,154.709
C04364=1062.867,-106.771,439.279,171.516,25.185,154.709
C04365=1062.874,-106.522,439.270,171.518,25.186,154.709
C04366=1062.879,-106.272,439.260,171.520,25.186,154.709
C04367=1062.885,-106.022,439.250,171.521,25.188,154.709
C04368=1062.892,-105.773,439.240,171.523,25.189,154.709
C04369=1062.898,-105.523,439.230,171.525,25.190,154.709
C04370=1062.903,-105.273,439.220,171.527,25.191,154.709
C04371=1062.910,-105.024,439.210,171.528,25.192,154.709
C04372=1062.916,-104.774,439.200,171.530,25.193,154.709
C04373=1062.922,-104.524,439.191,171.532,25.194,154.709
C04374=1062.928,-104.274,439.179,171.533,25.196,154.709
C04375=1062.935,-104.024,439.170,171.535,25.196,154.709
C04376=1062.941,-103.775,439.159,171.537,25.197,154.709
C04377=1062.946,-103.525,439.149,171.539,25.199,154.709
C04378=1062.953,-103.275,439.140,171.540,25.200,154.709
C04379=1062.959,-103.026,439.129,171.542,25.201,154.709
C04380=1062.965,-102.776,439.119,171.544,25.202,154.709
C04381=1062.971,-102.526,439.110,171.546,25.203,154.709
C04382=1062.977,-102.277,439.099,171.547,25.204,154.709
C04383=1062.983,-102.026,439.089,171.549,25.205,154.709
C04384=1062.990,-101.777,439.079,171.551,25.207,154.709
C04385=1062.996,-101.527,439.069,171.553,25.208,154.709
C04386=1063.002,-101.278,439.059,171.555,25.209,154.709
C04387=1063.008,-101.028,439.049,171.557,25.211,154.709
C04388=1063.014,-100.778,439.039,171.559,25.212,154.709
C04389=1063.020,-100.529,439.029,171.560,25.213,154.709
C04390=1063.026,-100.278,439.019,171.562,25.214,154.709
C04391=1063.032,-100.029,439.008,171.564,25.215,154.709
C04392=1063.038,-99.778,438.998,171.566,25.216,154.709
C04393=1063.045,-99.529,438.988,171.567,25.217,154.709
C04394=1063.051,-99.279,438.978,171.569,25.218,154.709
C04395=1063.057,-99.030,438.967,171.571,25.220,154.709
C04396=1063.064,-98.746,438.956,171.572,25.221,154.709
C04397=1063.071,-98.462,438.945,171.575,25.222,154.709
C04398=1063.078,-98.178,438.932,171.577,25.224,154.709
C04399=1063.086,-97.894,438.921,171.578,25.225,154.709
C04400=1063.091,-97.644,438.911,171.580,25.226,154.709
C04401=1063.098,-97.394,438.900,171.582,25.228,154.709
C04402=1063.103,-97.145,438.889,171.584,25.229,154.709
C04403=1063.109,-96.895,438.880,171.585,25.230,154.709
C04404=1063.115,-96.646,438.869,171.587,25.232,154.709
C04405=1063.122,-96.395,438.859,171.589,25.233,154.709
C04406=1063.128,-96.146,438.848,171.590,25.234,154.709
C04407=1063.134,-95.896,438.838,171.593,25.235,154.709
C04408=1063.140,-95.646,438.828,171.595,25.237,154.709
C04409=1063.145,-95.397,438.817,171.596,25.238,154.709
C04410=1063.152,-95.147,438.807,171.598,25.240,154.709
C04411=1063.158,-94.897,438.796,171.600,25.241,154.709
C04412=1063.164,-94.648,438.786,171.601,25.242,154.709
C04413=1063.170,-94.398,438.776,171.603,25.243,154.709
C04414=1063.176,-94.148,438.765,171.605,25.245,154.709
C04415=1063.182,-93.899,438.754,171.607,25.246,154.709
C04416=1063.187,-93.649,438.744,171.608,25.248,154.709
C04417=1063.194,-93.399,438.734,171.610,25.249,154.709
C04418=1063.200,-93.149,438.723,171.612,25.250,154.709
C04419=1063.206,-92.900,438.713,171.613,25.251,154.709
C04420=1063.212,-92.650,438.702,171.615,25.252,154.709
C04421=1063.218,-92.400,438.691,171.617,25.254,154.709
C04422=1063.225,-92.151,438.681,171.618,25.255,154.709
C04423=1063.230,-91.901,438.671,171.620,25.257,154.709
C04424=1063.237,-91.651,438.660,171.622,25.258,154.709
C04425=1063.243,-91.402,438.650,171.623,25.260,154.710
C04426=1063.249,-91.151,438.639,171.625,25.261,154.710
C04427=1063.255,-90.902,438.629,171.627,25.262,154.710
C04428=1063.261,-90.653,438.618,171.628,25.263,154.710
C04429=1063.267,-90.403,438.608,171.631,25.265,154.710
C04430=1063.274,-90.153,438.596,171.633,25.267,154.710
C04431=1063.279,-89.903,438.586,171.634,25.268,154.710
C04432=1063.286,-89.654,438.576,171.636,25.269,154.710
C04433=1063.292,-89.404,438.565,171.638,25.271,154.710
C04434=1063.298,-89.154,438.554,171.639,25.272,154.710
C04435=1063.304,-88.905,438.543,171.641,25.273,154.710
C04436=1063.310,-88.655,438.533,171.643,25.275,154.710
C04437=1063.316,-88.405,438.522,171.644,25.276,154.710
C04438=1063.322,-88.156,438.512,171.646,25.278,154.710
C04439=1063.328,-87.906,438.501,171.648,25.279,154.710
C04440=1063.334,-87.656,438.490,171.649,25.281,154.710
C04441=1063.341,-87.407,438.479,171.651,25.282,154.710
C04442=1063.346,-87.157,438.469,171.653,25.283,154.710
C04443=1063.353,-86.906,438.458,171.654,25.285,154.710
C04444=1063.359,-86.657,438.448,171.656,25.286,154.711
C04445=1063.365,-86.408,438.437,171.658,25.287,154.711
C04446=1063.371,-86.157,438.426,171.659,25.289,154.711
C04447=1063.378,-85.908,438.415,171.661,25.290,154.711
C04448=1063.384,-85.659,438.404,171.663,25.291,154.711
C04449=1063.390,-85.409,438.393,171.665,25.293,154.711
C04450=1063.396,-85.159,438.383,171.667,25.295,154.711
C04451=1063.402,-84.910,438.372,171.669,25.296,154.711
C04452=1063.408,-84.659,438.361,171.670,25.298,154.711
C04453=1063.415,-84.410,438.351,171.672,25.299,154.711
C04454=1063.420,-84.160,438.340,171.674,25.300,154.711
C04455=1063.427,-83.910,438.329,171.675,25.302,154.711
C04456=1063.433,-83.661,438.319,171.677,25.303,154.711
C04457=1063.439,-83.411,438.308,171.679,25.305,154.711
C04458=1063.445,-83.161,438.297,171.680,25.306,154.711
C04459=1063.452,-82.912,438.286,171.682,25.307,154.711
C04460=1063.458,-82.630,438.273,171.684,25.309,154.711
C04461=1063.466,-82.349,438.261,171.686,25.311,154.712
C04462=1063.473,-82.067,438.249,171.688,25.312,154.712
C04463=1063.479,-81.785,438.237,171.689,25.314,154.712
C04464=1063.486,-81.535,438.226,171.691,25.315,154.712
C04465=1063.492,-81.286,438.215,171.693,25.317,154.712
C04466=1063.499,-81.036,438.204,171.694,25.318,154.712
C04467=1063.504,-80.786,438.193,171.696,25.320,154.712
C04468=1063.511,-80.537,438.183,171.699,25.322,154.712
C04469=1063.517,-80.287,438.171,171.700,25.323,154.712
C04470=1063.523,-80.037,438.160,171.702,25.325,154.712
C04471=1063.529,-79.787,438.149,171.704,25.326,154.712
C04472=1063.535,-79.538,438.138,171.705,25.328,154.712
C04473=1063.542,-79.288,438.128,171.707,25.330,154.712
C04474=1063.548,-79.039,438.116,171.709,25.331,154.712
C04475=1063.554,-78.789,438.105,171.710,25.333,154.713
C04476=1063.560,-78.539,438.094,171.712,25.334,154.713
C04477=1063.566,-78.290,438.083,171.713,25.336,154.713
C04478=1063.572,-78.040,438.072,171.715,25.337,154.713
C04479=1063.578,-77.790,438.061,171.717,25.339,154.713
C04480=1063.584,-77.540,438.050,171.718,25.340,154.713
C04481=1063.590,-77.291,438.038,171.720,25.342,154.713
C04482=1063.596,-77.042,438.027,171.722,25.343,154.713
C04483=1063.602,-76.791,438.016,171.723,25.345,154.713
C04484=1063.608,-76.542,438.005,171.725,25.346,154.713
C04485=1063.614,-76.292,437.994,171.727,25.348,154.714
C04486=1063.621,-76.043,437.982,171.728,25.350,154.714
C04487=1063.627,-75.793,437.971,171.730,25.351,154.714
C04488=1063.633,-75.543,437.960,171.732,25.353,154.714
C04489=1063.639,-75.293,437.949,171.734,25.355,154.714
C04490=1063.645,-75.044,437.939,171.736,25.356,154.714
C04491=1063.652,-74.794,437.927,171.737,25.358,154.714
C04492=1063.658,-74.545,437.916,171.739,25.360,154.714
C04493=1063.664,-74.294,437.905,171.740,25.362,154.714
C04494=1063.670,-74.045,437.894,171.742,25.363,154.714
C04495=1063.677,-73.795,437.882,171.744,25.365,154.715
C04496=1063.682,-73.546,437.870,171.745,25.366,154.715
C04497=1063.687,-73.296,437.859,171.747,25.368,154.715
C04498=1063.694,-73.047,437.847,171.748,25.370,154.715
C04499=1063.700,-72.797,437.837,171.750,25.371,154.715
C04500=1063.706,-72.547,437.825,171.752,25.373,154.715
C04501=1063.711,-72.298,437.813,171.753,25.375,154.715
C04502=1063.718,-72.047,437.802,171.755,25.377,154.715
C04503=1063.723,-71.798,437.791,171.756,25.378,154.716
C04504=1063.730,-71.548,437.779,171.758,25.380,154.716
C04505=1063.736,-71.299,437.768,171.760,25.382,154.716
C04506=1063.742,-71.049,437.757,171.761,25.383,154.716
C04507=1063.747,-70.800,437.745,171.763,25.385,154.716
C04508=1063.754,-70.549,437.734,171.765,25.387,154.716
C04509=1063.760,-70.301,437.722,171.767,25.389,154.716
C04510=1063.766,-70.050,437.711,171.769,25.391,154.716
C04511=1063.771,-69.801,437.699,171.770,25.392,154.717
C04512=1063.778,-69.551,437.687,171.772,25.394,154.717
C04513=1063.784,-69.301,437.676,171.773,25.396,154.717
C04514=1063.790,-69.052,437.664,171.775,25.398,154.717
C04515=1063.796,-68.802,437.654,171.777,25.400,154.717
C04516=1063.802,-68.552,437.642,171.778,25.401,154.717
C04517=1063.808,-68.303,437.630,171.780,25.403,154.717
C04518=1063.814,-68.053,437.619,171.781,25.404,154.717
C04519=1063.820,-67.804,437.607,171.783,25.406,154.718
C04520=1063.826,-67.553,437.595,171.785,25.408,154.718
C04521=1063.832,-67.305,437.584,171.786,25.410,154.718
C04522=1063.838,-67.054,437.573,171.788,25.411,154.718
C04523=1063.844,-66.806,437.561,171.789,25.413,154.718
C04524=1063.851,-66.526,437.548,171.791,25.415,154.718
C04525=1063.858,-66.246,437.535,171.793,25.417,154.718
C04526=1063.865,-65.966,437.522,171.795,25.419,154.719
C04527=1063.872,-65.687,437.509,171.796,25.421,154.719
C04528=1063.877,-65.437,437.497,171.798,25.423,154.719
C04529=1063.883,-65.187,437.485,171.800,25.425,154.719
C04530=1063.889,-64.938,437.474,171.801,25.427,154.719
C04531=1063.896,-64.688,437.462,171.804,25.429,154.719
C04532=1063.901,-64.438,437.451,171.805,25.431,154.719
C04533=1063.907,-64.189,437.439,171.807,25.432,154.720
C04534=1063.914,-63.939,437.428,171.809,25.434,154.720
C04535=1063.920,-63.689,437.416,171.810,25.436,154.720
C04536=1063.926,-63.440,437.404,171.812,25.438,154.720
C04537=1063.932,-63.190,437.392,171.813,25.439,154.720
C04538=1063.938,-62.941,437.381,171.815,25.441,154.720
C04539=1063.944,-62.690,437.369,171.816,25.443,154.720
C04540=1063.950,-62.441,437.357,171.818,25.445,154.721
C04541=1063.956,-62.192,437.345,171.820,25.447,154.721
C04542=1063.963,-61.942,437.334,171.821,25.448,154.721
C04543=1063.968,-61.692,437.321,171.823,25.450,154.721
C04544=1063.975,-61.443,437.310,171.824,25.452,154.721
C04545=1063.981,-61.193,437.299,171.826,25.454,154.721
C04546=1063.987,-60.943,437.286,171.828,25.455,154.721
C04547=1063.993,-60.694,437.275,171.829,25.457,154.722
C04548=1063.999,-60.444,437.263,171.831,25.459,154.722
C04549=1064.005,-60.194,437.251,171.832,25.461,154.722
C04550=1064.011,-59.945,437.239,171.834,25.463,154.722
C04551=1064.017,-59.695,437.228,171.835,25.465,154.722
C04552=1064.023,-59.445,437.215,171.837,25.467,154.722
C04553=1064.030,-59.196,437.203,171.839,25.469,154.722
C04554=1064.036,-58.947,437.192,171.841,25.471,154.723
C04555=1064.042,-58.696,437.180,171.843,25.472,154.723
C04556=1064.048,-58.447,437.168,171.844,25.474,154.723
C04557=1064.054,-58.198,437.156,171.846,25.476,154.723
C04558=1064.060,-57.948,437.144,171.847,25.478,154.723
C04559=1064.067,-57.698,437.133,171.849,25.480,154.723
C04560=1064.073,-57.448,437.121,171.851,25.481,154.723
C04561=1064.079,-57.199,437.108,171.852,25.484,154.724
C04562=1064.085,-56.949,437.096,171.854,25.485,154.724
C04563=1064.092,-56.699,437.085,171.855,25.487,154.724
C04564=1064.097,-56.449,437.073,171.857,25.489,154.724
C04565=1064.104,-56.200,437.061,171.858,25.491,154.724
C04566=1064.110,-55.951,437.049,171.860,25.493,154.724
C04567=1064.116,-55.701,437.037,171.862,25.494,154.725
C04568=1064.123,-55.451,437.025,171.863,25.496,154.725
C04569=1064.128,-55.202,437.014,171.865,25.499,154.725
C04570=1064.134,-54.952,437.001,171.866,25.500,154.725
C04571=1064.141,-54.702,436.989,171.868,25.502,154.725
C04572=1064.147,-54.453,436.977,171.869,25.504,154.725
C04573=1064.154,-54.203,436.965,171.871,25.506,154.726
C04574=1064.160,-53.954,436.953,171.873,25.507,154.726
C04575=1064.166,-53.704,436.941,171.874,25.510,154.726
C04576=1064.172,-53.455,436.929,171.877,25.512,154.726
C04577=1064.178,-53.204,436.917,171.878,25.514,154.726
C04578=1064.184,-52.955,436.905,171.880,25.515,154.726
C04579=1064.191,-52.705,436.893,171.881,25.517,154.726
C04580=1064.196,-52.456,436.881,171.883,25.519,154.727
C04581=1064.203,-52.206,436.869,171.884,25.521,154.727
C04582=1064.209,-51.956,436.856,171.886,25.523,154.727
C04583=1064.216,-51.707,436.844,171.888,25.525,154.727
C04584=1064.222,-51.457,436.832,171.889,25.527,154.727
C04585=1064.228,-51.207,436.820,171.891,25.528,154.727
C04586=1064.235,-50.958,436.808,171.892,25.531,154.728
C04587=1064.240,-50.709,436.796,171.894,25.533,154.728
C04588=1064.248,-50.430,436.782,171.895,25.534,154.728
C04589=1064.255,-50.152,436.769,171.898,25.537,154.728
C04590=1064.262,-49.874,436.755,171.899,25.539,154.729
C04591=1064.268,-49.595,436.741,171.901,25.541,154.729
C04592=1064.274,-49.346,436.729,171.902,25.543,154.729
C04593=1064.280,-49.096,436.716,171.904,25.545,154.729
C04594=1064.285,-48.847,436.704,171.905,25.547,154.729
C04595=1064.292,-48.597,436.692,171.907,25.549,154.729
C04596=1064.298,-48.347,436.679,171.908,25.551,154.730
C04597=1064.304,-48.097,436.667,171.910,25.554,154.730
C04598=1064.310,-47.848,436.655,171.912,25.555,154.730
C04599=1064.316,-47.598,436.643,171.913,25.558,154.730
C04600=1064.322,-47.349,436.629,171.915,25.559,154.730
C04601=1064.329,-47.100,436.618,171.916,25.561,154.731
C04602=1064.334,-46.850,436.605,171.918,25.564,154.731
C04603=1064.340,-46.600,436.592,171.919,25.565,154.731
C04604=1064.346,-46.350,436.580,171.921,25.568,154.731
C04605=1064.352,-46.101,436.568,171.923,25.570,154.731
C04606=1064.358,-45.851,436.556,171.925,25.572,154.732
C04607=1064.364,-45.601,436.543,171.926,25.574,154.732
C04608=1064.370,-45.352,436.530,171.928,25.576,154.732
C04609=1064.377,-45.102,436.518,171.929,25.578,154.732
C04610=1064.383,-44.853,436.505,171.931,25.580,154.732
C04611=1064.389,-44.603,436.493,171.932,25.582,154.733
C04612=1064.395,-44.353,436.480,171.934,25.584,154.733
C04613=1064.401,-44.103,436.468,171.935,25.586,154.733
C04614=1064.407,-43.855,436.455,171.937,25.588,154.733
C04615=1064.413,-43.605,436.443,171.939,25.590,154.733
C04616=1064.419,-43.355,436.430,171.940,25.592,154.734
C04617=1064.425,-43.105,436.418,171.942,25.595,154.734
C04618=1064.431,-42.855,436.406,171.943,25.596,154.734
C04619=1064.438,-42.606,436.393,171.945,25.599,154.734
C04620=1064.443,-42.356,436.380,171.946,25.600,154.734
C04621=1064.450,-42.107,436.368,171.948,25.603,154.735
C04622=1064.456,-41.857,436.355,171.949,25.605,154.735
C04623=1064.462,-41.608,436.342,171.951,25.607,154.735
C04624=1064.468,-41.358,436.330,171.952,25.609,154.735
C04625=1064.475,-41.108,436.318,171.954,25.611,154.735
C04626=1064.481,-40.859,436.304,171.955,25.613,154.736
C04627=1064.487,-40.609,436.292,171.957,25.615,154.736
C04628=1064.493,-40.359,436.279,171.958,25.617,154.736
C04629=1064.498,-40.111,436.266,171.960,25.619,154.736
C04630=1064.505,-39.861,436.254,171.961,25.622,154.737
C04631=1064.511,-39.611,436.242,171.963,25.623,154.737
C04632=1064.517,-39.361,436.229,171.964,25.626,154.737
C04633=1064.523,-39.112,436.216,171.966,25.628,154.737
C04634=1064.529,-38.862,436.203,171.968,25.630,154.737
C04635=1064.536,-38.613,436.191,171.969,25.632,154.737
C04636=1064.542,-38.363,436.178,171.971,25.634,154.738
C04637=1064.548,-38.113,436.166,171.972,25.636,154.738
C04638=1064.554,-37.864,436.152,171.974,25.638,154.738
C04639=1064.560,-37.614,436.140,171.975,25.640,154.738
C04640=1064.566,-37.364,436.127,171.978,25.643,154.739
C04641=1064.572,-37.115,436.114,171.979,25.645,154.739
C04642=1064.578,-36.865,436.102,171.981,25.647,154.739
C04643=1064.584,-36.616,436.088,171.982,25.650,154.739
C04644=1064.590,-36.366,436.076,171.984,25.651,154.739
C04645=1064.596,-36.117,436.062,171.985,25.654,154.740
C04646=1064.602,-35.867,436.050,171.987,25.656,154.740
C04647=1064.608,-35.617,436.037,171.988,25.658,154.740
C04648=1064.614,-35.368,436.024,171.990,25.660,154.740
C04649=1064.620,-35.118,436.011,171.991,25.662,154.741
C04650=1064.626,-34.869,435.998,171.993,25.664,154.741
C04651=1064.632,-34.619,435.986,171.994,25.667,154.741
C04652=1064.639,-34.341,435.971,171.996,25.669,154.741
C04653=1064.645,-34.063,435.957,171.997,25.671,154.742
C04654=1064.653,-33.786,435.942,171.999,25.674,154.742
C04655=1064.659,-33.508,435.927,172.001,25.676,154.742
C04656=1064.665,-33.258,435.915,172.002,25.679,154.742
C04657=1064.671,-33.009,435.901,172.004,25.681,154.743
C04658=1064.677,-32.758,435.888,172.006,25.683,154.743
C04659=1064.684,-32.509,435.875,172.007,25.685,154.743
C04660=1064.690,-32.259,435.863,172.008,25.687,154.743
C04661=1064.696,-32.010,435.849,172.010,25.690,154.744
C04662=1064.702,-31.760,435.837,172.012,25.692,154.744
C04663=1064.708,-31.511,435.823,172.013,25.694,154.744
C04664=1064.714,-31.261,435.810,172.014,25.696,154.744
C04665=1064.720,-31.011,435.798,172.016,25.699,154.745
C04666=1064.726,-30.762,435.784,172.018,25.700,154.745
C04667=1064.732,-30.512,435.772,172.019,25.703,154.745
C04668=1064.738,-30.263,435.759,172.020,25.705,154.745
C04669=1064.745,-30.014,435.745,172.022,25.707,154.745
C04670=1064.751,-29.764,435.733,172.024,25.709,154.746
C04671=1064.757,-29.514,435.719,172.025,25.711,154.746
C04672=1064.763,-29.264,435.705,172.026,25.714,154.746
C04673=1064.769,-29.014,435.693,172.028,25.716,154.746
C04674=1064.775,-28.765,435.679,172.030,25.718,154.747
C04675=1064.781,-28.516,435.666,172.031,25.720,154.747
C04676=1064.787,-28.266,435.654,172.033,25.723,154.747
C04677=1064.793,-28.017,435.640,172.034,25.725,154.747
C04678=1064.799,-27.767,435.627,172.036,25.727,154.748
C04679=1064.806,-27.517,435.614,172.037,25.729,154.748
C04680=1064.812,-27.268,435.601,172.039,25.731,154.748
C04681=1064.818,-27.018,435.588,172.040,25.734,154.748
C04682=1064.825,-26.769,435.574,172.041,25.736,154.749
C04683=1064.830,-26.519,435.561,172.043,25.738,154.749
C04684=1064.836,-26.270,435.548,172.045,25.740,154.749
C04685=1064.842,-26.020,435.535,172.046,25.743,154.749
C04686=1064.848,-25.771,435.521,172.048,25.745,154.750
C04687=1064.854,-25.520,435.508,172.049,25.747,154.750
C04688=1064.860,-25.271,435.495,172.050,25.750,154.750
C04689=1064.866,-25.021,435.481,172.052,25.752,154.750
C04690=1064.872,-24.772,435.467,172.053,25.754,154.751
C04691=1064.878,-24.523,435.454,172.055,25.757,154.751
C04692=1064.884,-24.273,435.442,172.056,25.759,154.751
C04693=1064.890,-24.023,435.428,172.058,25.761,154.751
C04694=1064.897,-23.773,435.414,172.059,25.764,154.752
C04695=1064.903,-23.524,435.401,172.061,25.765,154.752
C04696=1064.908,-23.275,435.387,172.062,25.768,154.752
C04697=1064.914,-23.025,435.374,172.064,25.770,154.752
C04698=1064.920,-22.775,435.361,172.065,25.772,154.753
C04699=1064.926,-22.526,435.347,172.067,25.775,154.753
C04700=1064.933,-22.276,435.334,172.068,25.777,154.753
C04701=1064.939,-22.027,435.320,172.070,25.779,154.753
C04702=1064.944,-21.777,435.306,172.071,25.782,154.754
C04703=1064.951,-21.528,435.293,172.073,25.784,154.754
C04704=1064.957,-21.279,435.280,172.074,25.786,154.754
C04705=1064.962,-21.029,435.266,172.076,25.789,154.755
C04706=1064.969,-20.779,435.252,172.077,25.791,154.755
C04707=1064.975,-20.529,435.240,172.079,25.793,154.755
C04708=1064.980,-20.280,435.226,172.080,25.796,154.755
C04709=1064.987,-20.030,435.213,172.082,25.798,154.756
C04710=1064.993,-19.780,435.199,172.083,25.800,154.756
C04711=1064.999,-19.531,435.185,172.085,25.803,154.756
C04712=1065.005,-19.281,435.172,172.086,25.805,154.756
C04713=1065.011,-19.032,435.159,172.087,25.807,154.757
C04714=1065.017,-18.783,435.145,172.089,25.810,154.757
C04715=1065.024,-18.533,435.131,172.090,25.812,154.757
C04716=1065.030,-18.254,435.116,172.093,25.815,154.757
C04717=1065.037,-17.975,435.101,172.094,25.817,154.758
C04718=1065.044,-17.696,435.086,172.096,25.820,154.758
C04719=1065.051,-17.418,435.070,172.097,25.822,154.758
C04720=1065.057,-17.169,435.057,172.099,25.825,154.759
C04721=1065.063,-16.919,435.043,172.100,25.827,154.759
C04722=1065.069,-16.670,435.030,172.102,25.829,154.759
C04723=1065.075,-16.420,435.015,172.103,25.832,154.759
C04724=1065.081,-16.171,435.002,172.105,25.834,154.760
C04725=1065.087,-15.921,434.989,172.106,25.836,154.760
C04726=1065.094,-15.671,434.975,172.108,25.839,154.760
C04727=1065.100,-15.422,434.961,172.109,25.841,154.760
C04728=1065.105,-15.172,434.947,172.110,25.843,154.761
C04729=1065.112,-14.922,434.934,172.112,25.846,154.761
C04730=1065.118,-14.673,434.920,172.113,25.848,154.761
C04731=1065.124,-14.423,434.907,172.115,25.850,154.762
C04732=1065.130,-14.175,434.892,172.116,25.853,154.762
C04733=1065.136,-13.925,434.878,172.118,25.855,154.762
C04734=1065.142,-13.675,434.865,172.119,25.857,154.762
C04735=1065.147,-13.425,434.851,172.121,25.860,154.763
C04736=1065.153,-13.176,434.837,172.122,25.862,154.763
C04737=1065.160,-12.926,434.823,172.124,25.865,154.763
C04738=1065.166,-12.677,434.809,172.125,25.867,154.764
C04739=1065.172,-12.428,434.795,172.127,25.869,154.764
C04740=1065.178,-12.177,434.781,172.128,25.872,154.764
C04741=1065.184,-11.928,434.768,172.130,25.874,154.764
C04742=1065.189,-11.679,434.754,172.131,25.876,154.765
C04743=1065.196,-11.429,434.740,172.132,25.879,154.765
C04744=1065.202,-11.180,434.726,172.134,25.882,154.765
C04745=1065.207,-10.930,434.712,172.135,25.884,154.766
C04746=1065.214,-10.680,434.698,172.137,25.886,154.766
C04747=1065.220,-10.430,434.684,172.138,25.889,154.766
C04748=1065.225,-10.182,434.670,172.140,25.891,154.766
C04749=1065.232,-9.932,434.656,172.141,25.893,154.767
C04750=1065.238,-9.682,434.642,172.143,25.896,154.767
C04751=1065.244,-9.433,434.628,172.144,25.899,154.767
C04752=1065.250,-9.183,434.614,172.146,25.901,154.768
C04753=1065.256,-8.933,434.600,172.147,25.903,154.768
C04754=1065.262,-8.684,434.587,172.149,25.906,154.768
C04755=1065.268,-8.435,434.572,172.150,25.908,154.768
C04756=1065.274,-8.185,434.558,172.152,25.910,154.769
C04757=1065.280,-7.936,434.545,172.153,25.913,154.769
C04758=1065.287,-7.686,434.530,172.155,25.915,154.769
C04759=1065.292,-7.437,434.516,172.156,25.918,154.770
C04760=1065.299,-7.187,434.503,172.157,25.920,154.770
C04761=1065.305,-6.938,434.488,172.159,25.922,154.770
C04762=1065.310,-6.688,434.474,172.160,25.925,154.770
C04763=1065.317,-6.438,434.460,172.162,25.928,154.771
C04764=1065.323,-6.189,434.446,172.163,25.930,154.771
C04765=1065.329,-5.939,434.432,172.165,25.932,154.771
C04766=1065.335,-5.690,434.418,172.166,25.935,154.772
C04767=1065.341,-5.440,434.403,172.168,25.937,154.772
C04768=1065.347,-5.190,434.390,172.169,25.939,154.772
C04769=1065.353,-4.942,434.376,172.171,25.942,154.773
C04770=1065.359,-4.691,434.361,172.172,25.944,154.773
C04771=1065.365,-4.442,434.347,172.174,25.947,154.773
C04772=1065.372,-4.192,434.333,172.175,25.949,154.773
C04773=1065.378,-3.944,434.319,172.177,25.951,154.774
C04774=1065.384,-3.693,434.304,172.178,25.954,154.774
C04775=1065.390,-3.444,434.291,172.179,25.957,154.774
C04776=1065.396,-3.194,434.276,172.181,25.959,154.775
C04777=1065.402,-2.945,434.262,172.182,25.961,154.775
C04778=1065.408,-2.696,434.248,172.184,25.964,154.775
C04779=1065.414,-2.446,434.233,172.184,25.966,154.776
C04780=1065.420,-2.166,434.217,172.187,25.969,154.776
C04781=1065.428,-1.885,434.201,172.188,25.972,154.776
C04782=1065.434,-1.605,434.184,172.189,25.975,154.777
C04783=1065.440,-1.325,434.169,172.191,25.978,154.777
C04784=1065.446,-1.075,434.154,172.192,25.980,154.777
C04785=1065.452,-0.826,434.140,172.194,25.982,154.777
C04786=1065.458,-0.576,434.125,172.195,25.985,154.778
C04787=1065.464,-0.327,434.110,172.197,25.987,154.778
C04788=1065.470,-0.078,434.097,172.198,25.990,154.779
C04789=1065.477,0.172,434.082,172.200,25.993,154.779
C04790=1065.482,0.422,434.068,172.201,25.995,154.779
C04791=1065.488,0.671,434.053,172.202,25.998,154.779
C04792=1065.494,0.921,434.040,172.204,26.000,154.780
C04793=1065.500,1.170,434.025,172.205,26.002,154.780
C04794=1065.506,1.419,434.010,172.207,26.005,154.780
C04795=1065.512,1.670,433.996,172.208,26.008,154.781
C04796=1065.518,1.919,433.981,172.210,26.010,154.781
C04797=1065.524,2.168,433.966,172.211,26.013,154.781
C04798=1065.530,2.418,433.952,172.213,26.015,154.782
C04799=1065.536,2.668,433.937,172.214,26.018,154.782
C04800=1065.542,2.916,433.923,172.215,26.020,154.782
C04801=1065.548,3.167,433.909,172.217,26.023,154.783
C04802=1065.554,3.416,433.894,172.218,26.025,154.783
C04803=1065.560,3.665,433.879,172.220,26.028,154.783
C04804=1065.566,3.915,433.865,172.221,26.030,154.783
C04805=1065.572,4.165,433.850,172.223,26.033,154.784
C04806=1065.578,4.414,433.836,172.224,26.036,154.784
C04807=1065.584,4.664,433.822,172.226,26.038,154.784
C04808=1065.590,4.913,433.807,172.227,26.041,154.785
C04809=1065.596,5.162,433.792,172.229,26.043,154.785
C04810=1065.602,5.411,433.777,172.230,26.045,154.785
C04811=1065.608,5.662,433.763,172.231,26.048,154.786
C04812=1065.614,5.911,433.749,172.233,26.051,154.786
C04813=1065.620,6.160,433.734,172.233,26.053,154.786
C04814=1065.626,6.410,433.719,172.235,26.055,154.787
C04815=1065.632,6.660,433.705,172.236,26.058,154.787
C04816=1065.638,6.910,433.689,172.238,26.060,154.787
C04817=1065.643,7.158,433.675,172.239,26.063,154.788
C04818=1065.650,7.408,433.660,172.241,26.065,154.788
C04819=1065.656,7.657,433.645,172.242,26.068,154.788
C04820=1065.662,7.907,433.630,172.244,26.071,154.789
C04821=1065.668,8.157,433.616,172.245,26.073,154.789
C04822=1065.674,8.406,433.601,172.246,26.076,154.789
C04823=1065.680,8.656,433.587,172.248,26.078,154.789
C04824=1065.686,8.905,433.572,172.249,26.080,154.790
C04825=1065.692,9.154,433.557,172.251,26.083,154.790
C04826=1065.699,9.404,433.542,172.252,26.086,154.790
C04827=1065.704,9.653,433.528,172.254,26.088,154.791
C04828=1065.711,9.903,433.513,172.255,26.091,154.791
C04829=1065.717,10.153,433.498,172.257,26.093,154.791
C04830=1065.723,10.402,433.484,172.258,26.096,154.792
C04831=1065.729,10.651,433.469,172.260,26.098,154.792
C04832=1065.735,10.901,433.454,172.261,26.101,154.792
C04833=1065.741,11.150,433.439,172.262,26.103,154.793
C04834=1065.747,11.400,433.424,172.264,26.106,154.793
C04835=1065.753,11.649,433.409,172.265,26.108,154.793
C04836=1065.759,11.899,433.394,172.267,26.111,154.794
C04837=1065.765,12.148,433.379,172.268,26.113,154.794
C04838=1065.772,12.398,433.364,172.270,26.116,154.794
C04839=1065.778,12.647,433.350,172.271,26.118,154.795
C04840=1065.784,12.896,433.335,172.273,26.121,154.795
C04841=1065.790,13.147,433.321,172.274,26.124,154.795
C04842=1065.796,13.396,433.306,172.276,26.126,154.796
C04843=1065.802,13.645,433.291,172.276,26.128,154.796
C04844=1065.809,13.927,433.274,172.279,26.131,154.796
C04845=1065.816,14.209,433.257,172.280,26.134,154.797
C04846=1065.823,14.492,433.239,172.281,26.137,154.797
C04847=1065.830,14.774,433.223,172.283,26.140,154.797
C04848=1065.835,15.023,433.208,172.284,26.142,154.798
C04849=1065.842,15.273,433.193,172.286,26.145,154.798
C04850=1065.847,15.523,433.177,172.287,26.147,154.798
C04851=1065.853,15.772,433.163,172.288,26.150,154.799
C04852=1065.860,16.022,433.148,172.290,26.153,154.799
C04853=1065.865,16.272,433.132,172.291,26.155,154.799
C04854=1065.871,16.520,433.117,172.293,26.158,154.800
C04855=1065.878,16.769,433.102,172.294,26.161,154.800
C04856=1065.883,17.019,433.087,172.296,26.163,154.800
C04857=1065.889,17.268,433.072,172.297,26.166,154.801
C04858=1065.895,17.518,433.057,172.299,26.168,154.801
C04859=1065.901,17.768,433.042,172.300,26.171,154.801
C04860=1065.907,18.018,433.027,172.301,26.173,154.802
C04861=1065.913,18.267,433.012,172.303,26.176,154.802
C04862=1065.919,18.516,432.996,172.304,26.178,154.802
C04863=1065.926,18.766,432.981,172.306,26.181,154.803
C04864=1065.931,19.015,432.966,172.307,26.184,154.803
C04865=1065.937,19.265,432.951,172.309,26.187,154.803
C04866=1065.943,19.514,432.936,172.310,26.189,154.804
C04867=1065.950,19.764,432.921,172.312,26.192,154.804
C04868=1065.955,20.013,432.905,172.313,26.194,154.804
C04869=1065.962,20.262,432.890,172.313,26.197,154.805
C04870=1065.968,20.512,432.875,172.315,26.199,154.805
C04871=1065.974,20.762,432.859,172.316,26.202,154.805
C04872=1065.980,21.010,432.844,172.318,26.204,154.806
C04873=1065.985,21.260,432.829,172.319,26.207,154.806
C04874=1065.992,21.510,432.814,172.321,26.209,154.806
C04875=1065.997,21.760,432.798,172.322,26.212,154.807
C04876=1066.003,22.008,432.783,172.324,26.214,154.807
C04877=1066.009,22.258,432.767,172.325,26.217,154.807
C04878=1066.015,22.508,432.752,172.326,26.220,154.808
C04879=1066.021,22.758,432.737,172.328,26.223,154.808
C04880=1066.027,23.006,432.722,172.329,26.225,154.808
C04881=1066.033,23.256,432.706,172.331,26.228,154.809
C04882=1066.039,23.506,432.691,172.332,26.231,154.809
C04883=1066.045,23.755,432.675,172.334,26.233,154.809
C04884=1066.052,24.005,432.660,172.335,26.236,154.810
C04885=1066.057,24.254,432.645,172.337,26.238,154.810
C04886=1066.063,24.503,432.629,172.338,26.241,154.810
C04887=1066.070,24.753,432.614,172.339,26.244,154.811
C04888=1066.075,25.003,432.599,172.341,26.246,154.811
C04889=1066.082,25.252,432.583,172.342,26.249,154.812
C04890=1066.087,25.501,432.568,172.344,26.251,154.812
C04891=1066.094,25.750,432.552,172.344,26.254,154.812
C04892=1066.099,26.000,432.536,172.346,26.256,154.812
C04893=1066.105,26.250,432.521,172.347,26.259,154.813
C04894=1066.112,26.499,432.505,172.349,26.261,154.813
C04895=1066.117,26.748,432.490,172.350,26.264,154.814
C04896=1066.123,26.997,432.474,172.352,26.267,154.814
C04897=1066.129,27.247,432.459,172.353,26.269,154.814
C04898=1066.135,27.497,432.444,172.354,26.272,154.815
C04899=1066.141,27.746,432.428,172.356,26.275,154.815
C04900=1066.148,27.996,432.413,172.357,26.277,154.815
C04901=1066.154,28.245,432.396,172.359,26.280,154.816
C04902=1066.160,28.494,432.382,172.360,26.283,154.816
C04903=1066.165,28.743,432.366,172.362,26.285,154.816
C04904=1066.171,28.993,432.350,172.363,26.288,154.817
C04905=1066.178,29.242,432.334,172.365,26.291,154.817
C04906=1066.183,29.492,432.319,172.366,26.293,154.817
C04907=1066.189,29.742,432.303,172.367,26.296,154.818
C04908=1066.196,30.025,432.285,172.369,26.299,154.818
C04909=1066.203,30.308,432.267,172.370,26.302,154.818
C04910=1066.210,30.592,432.249,172.372,26.304,154.819
C04911=1066.216,30.876,432.232,172.374,26.308,154.819
C04912=1066.222,31.125,432.216,172.375,26.311,154.820
C04913=1066.228,31.374,432.200,172.377,26.313,154.820
C04914=1066.234,31.624,432.184,172.377,26.315,154.820
C04915=1066.240,31.874,432.169,172.379,26.318,154.821
C04916=1066.246,32.123,432.153,172.380,26.321,154.821
C04917=1066.251,32.372,432.137,172.382,26.323,154.821
C04918=1066.258,32.621,432.122,172.383,26.326,154.822
C04919=1066.264,32.871,432.106,172.384,26.329,154.822
C04920=1066.270,33.120,432.090,172.386,26.331,154.822
C04921=1066.275,33.370,432.074,172.387,26.334,154.823
C04922=1066.282,33.619,432.059,172.389,26.337,154.823
C04923=1066.288,33.869,432.042,172.390,26.339,154.824
C04924=1066.294,34.119,432.027,172.392,26.342,154.824
C04925=1066.300,34.368,432.010,172.393,26.345,154.824
C04926=1066.306,34.617,431.995,172.395,26.348,154.825
C04927=1066.312,34.867,431.979,172.396,26.350,154.825
C04928=1066.318,35.117,431.963,172.398,26.353,154.825
C04929=1066.323,35.365,431.947,172.399,26.356,154.826
C04930=1066.330,35.615,431.932,172.400,26.358,154.826
C04931=1066.336,35.864,431.916,172.402,26.361,154.826
C04932=1066.342,36.113,431.900,172.403,26.364,154.827
C04933=1066.348,36.363,431.883,172.405,26.366,154.827
C04934=1066.354,36.612,431.868,172.406,26.369,154.827
C04935=1066.360,36.862,431.852,172.408,26.372,154.828
C04936=1066.366,37.111,431.836,172.408,26.374,154.828
C04937=1066.372,37.361,431.820,172.410,26.376,154.828
C04938=1066.377,37.611,431.804,172.411,26.379,154.829
C04939=1066.384,37.860,431.789,172.412,26.382,154.829
C04940=1066.390,38.109,431.772,172.414,26.385,154.830
C04941=1066.396,38.358,431.756,172.415,26.387,154.830
C04942=1066.402,38.608,431.740,172.417,26.390,154.830
C04943=1066.408,38.858,431.724,172.418,26.393,154.831
C04944=1066.414,39.107,431.708,172.420,26.395,154.831
C04945=1066.420,39.356,431.692,172.421,26.398,154.831
C04946=1066.425,39.606,431.675,172.423,26.401,154.832
C04947=1066.431,39.855,431.659,172.424,26.403,154.832
C04948=1066.437,40.105,431.644,172.425,26.406,154.832
C04949=1066.443,40.354,431.627,172.427,26.409,154.833
C04950=1066.449,40.604,431.611,172.428,26.411,154.833
C04951=1066.455,40.853,431.595,172.430,26.414,154.833
C04952=1066.461,41.102,431.579,172.431,26.417,154.834
C04953=1066.467,41.352,431.562,172.433,26.419,154.834
C04954=1066.473,41.601,431.546,172.434,26.422,154.835
C04955=1066.479,41.850,431.530,172.436,26.425,154.835
C04956=1066.484,42.100,431.514,172.437,26.427,154.835
C04957=1066.490,42.350,431.498,172.437,26.430,154.836
C04958=1066.496,42.599,431.482,172.439,26.432,154.836
C04959=1066.502,42.848,431.466,172.440,26.435,154.836
C04960=1066.508,43.098,431.449,172.442,26.438,154.837
C04961=1066.514,43.347,431.433,172.443,26.440,154.837
C04962=1066.520,43.596,431.417,172.445,26.443,154.837
C04963=1066.526,43.846,431.400,172.446,26.446,154.838
C04964=1066.532,44.095,431.384,172.447,26.449,154.838
C04965=1066.538,44.344,431.368,172.449,26.451,154.839
C04966=1066.544,44.594,431.352,172.450,26.454,154.839
C04967=1066.550,44.843,431.335,172.452,26.457,154.839
C04968=1066.555,45.093,431.319,172.453,26.460,154.840
C04969=1066.561,45.342,431.302,172.455,26.463,154.840
C04970=1066.567,45.592,431.286,172.456,26.465,154.840
C04971=1066.573,45.841,431.270,172.458,26.468,154.841
C04972=1066.579,46.124,431.251,172.459,26.471,154.841
C04973=1066.586,46.408,431.232,172.460,26.474,154.842
C04974=1066.593,46.691,431.214,172.462,26.477,154.842
C04975=1066.599,46.975,431.195,172.464,26.481,154.843
C04976=1066.605,47.224,431.179,172.465,26.483,154.843
C04977=1066.611,47.473,431.163,172.467,26.486,154.843
C04978=1066.616,47.723,431.146,172.468,26.489,154.844
C04979=1066.623,47.973,431.129,172.470,26.491,154.844
C04980=1066.629,48.222,431.112,172.470,26.493,154.844
C04981=1066.635,48.471,431.096,172.472,26.496,154.845
C04982=1066.640,48.721,431.079,172.473,26.499,154.845
C04983=1066.646,48.970,431.063,172.475,26.502,154.846
C04984=1066.652,49.219,431.047,172.476,26.505,154.846
C04985=1066.658,49.469,431.030,172.477,26.507,154.846
C04986=1066.663,49.719,431.014,172.479,26.510,154.847
C04987=1066.669,49.967,430.997,172.480,26.513,154.847
C04988=1066.675,50.217,430.980,172.482,26.516,154.847
C04989=1066.681,50.466,430.964,172.483,26.518,154.848
C04990=1066.687,50.715,430.948,172.485,26.521,154.848
C04991=1066.693,50.965,430.931,172.486,26.524,154.848
C04992=1066.699,51.215,430.914,172.488,26.527,154.849
C04993=1066.705,51.464,430.897,172.489,26.529,154.849
C04994=1066.711,51.713,430.881,172.490,26.532,154.850
C04995=1066.717,51.963,430.864,172.492,26.535,154.850
C04996=1066.722,52.212,430.848,172.493,26.537,154.850
C04997=1066.729,52.461,430.831,172.495,26.540,154.851
C04998=1066.734,52.710,430.814,172.496,26.543,154.851
C04999=1066.740,52.961,430.798,172.498,26.545,154.851
C05000=1066.746,53.210,430.781,172.499,26.548,154.852
C05001=1066.753,53.459,430.764,172.500,26.551,154.852
C05002=1066.758,53.708,430.747,172.502,26.553,154.852
C05003=1066.764,53.958,430.731,172.503,26.556,154.853
C05004=1066.770,54.206,430.714,172.504,26.559,154.853
C05005=1066.775,54.456,430.697,172.505,26.562,154.854
C05006=1066.782,54.706,430.681,172.507,26.564,154.854
C05007=1066.788,54.955,430.664,172.508,26.567,154.854
C05008=1066.794,55.204,430.648,172.510,26.570,154.855
C05009=1066.799,55.454,430.631,172.511,26.573,154.855
C05010=1066.806,55.702,430.614,172.513,26.575,154.855
C05011=1066.812,55.953,430.597,172.514,26.578,154.856
C05012=1066.817,56.202,430.580,172.516,26.580,154.856
C05013=1066.824,56.451,430.563,172.517,26.583,154.857
C05014=1066.830,56.700,430.547,172.518,26.586,154.857
C05015=1066.835,56.950,430.530,172.520,26.588,154.857
C05016=1066.842,57.199,430.513,172.521,26.591,154.858
C05017=1066.848,57.449,430.497,172.523,26.594,154.858
C05018=1066.854,57.697,430.480,172.524,26.596,154.858
C05019=1066.859,57.947,430.463,172.526,26.599,154.859
C05020=1066.866,58.197,430.446,172.527,26.602,154.859
C05021=1066.872,58.446,430.429,172.529,26.604,154.859
C05022=1066.877,58.696,430.412,172.530,26.607,154.860
C05023=1066.883,58.944,430.395,172.532,26.610,154.860
C05024=1066.890,59.194,430.379,172.533,26.612,154.861
C05025=1066.895,59.443,430.361,172.534,26.615,154.861
C05026=1066.901,59.693,430.345,172.536,26.618,154.861
C05027=1066.908,59.942,430.328,172.537,26.620,154.862
C05028=1066.913,60.192,430.311,172.539,26.623,154.862
C05029=1066.920,60.441,430.294,172.540,26.626,154.862
C05030=1066.925,60.690,430.277,172.542,26.629,154.863
C05031=1066.932,60.940,430.260,172.543,26.631,154.863
C05032=1066.938,61.189,430.243,172.545,26.634,154.863
C05033=1066.943,61.438,430.226,172.545,26.637,154.864
C05034=1066.950,61.688,430.209,172.547,26.639,154.864
C05035=1066.956,61.937,430.192,172.548,26.642,154.865
C05036=1066.963,62.220,430.173,172.550,26.645,154.865
C05037=1066.970,62.504,430.153,172.552,26.648,154.865
C05038=1066.976,62.787,430.134,172.553,26.651,154.866
C05039=1066.983,63.070,430.115,172.555,26.654,154.866
C05040=1066.990,63.320,430.098,172.556,26.656,154.867
C05041=1066.995,63.569,430.080,172.558,26.659,154.867
C05042=1067.001,63.818,430.064,172.559,26.662,154.867
C05043=1067.008,64.068,430.047,172.561,26.664,154.868
C05044=1067.013,64.317,430.029,172.562,26.667,154.868
C05045=1067.019,64.566,430.013,172.563,26.670,154.868
C05046=1067.025,64.816,429.995,172.565,26.673,154.869
C05047=1067.031,65.065,429.979,172.566,26.675,154.869
C05048=1067.037,65.314,429.961,172.568,26.678,154.870
C05049=1067.043,65.564,429.943,172.569,26.681,154.870
C05050=1067.049,65.813,429.927,172.571,26.683,154.870
C05051=1067.054,66.062,429.909,172.572,26.686,154.871
C05052=1067.061,66.312,429.892,172.574,26.689,154.871
C05053=1067.067,66.561,429.874,172.575,26.691,154.871
C05054=1067.072,66.810,429.858,172.577,26.694,154.872
C05055=1067.079,67.060,429.840,172.578,26.697,154.872
C05056=1067.084,67.309,429.823,172.579,26.700,154.873
C05057=1067.090,67.558,429.806,172.581,26.702,154.873
C05058=1067.097,67.808,429.788,172.582,26.705,154.873
C05059=1067.102,68.057,429.771,172.584,26.708,154.874
C05060=1067.108,68.306,429.754,172.585,26.711,154.874
C05061=1067.114,68.556,429.737,172.587,26.713,154.874
C05062=1067.120,68.805,429.719,172.588,26.716,154.875
C05063=1067.126,69.054,429.702,172.590,26.719,154.875
C05064=1067.132,69.304,429.684,172.591,26.722,154.876
C05065=1067.138,69.553,429.667,172.593,26.724,154.876
C05066=1067.144,69.803,429.650,172.594,26.727,154.876
C05067=1067.150,70.052,429.632,172.596,26.729,154.877
C05068=1067.155,70.301,429.615,172.597,26.732,154.877
C05069=1067.161,70.550,429.597,172.598,26.735,154.877
C05070=1067.167,70.800,429.579,172.600,26.738,154.878
C05071=1067.173,71.048,429.562,172.601,26.740,154.878
C05072=1067.179,71.299,429.545,172.603,26.743,154.878
C05073=1067.184,71.548,429.528,172.604,26.746,154.879
C05074=1067.190,71.797,429.510,172.606,26.749,154.879
C05075=1067.197,72.046,429.493,172.607,26.752,154.880
C05076=1067.202,72.295,429.475,172.609,26.754,154.880
C05077=1067.208,72.545,429.457,172.610,26.757,154.880
C05078=1067.214,72.794,429.440,172.612,26.760,154.881
C05079=1067.219,73.043,429.422,172.613,26.762,154.881
C05080=1067.226,73.292,429.405,172.613,26.765,154.882
C05081=1067.232,73.541,429.387,172.615,26.768,154.882
C05082=1067.238,73.792,429.370,172.616,26.770,154.882
C05083=1067.243,74.041,429.352,172.618,26.773,154.883
C05084=1067.249,74.291,429.334,172.619,26.776,154.883
C05085=1067.255,74.540,429.317,172.621,26.779,154.883
C05086=1067.261,74.788,429.300,172.622,26.781,154.884
C05087=1067.267,75.038,429.282,172.624,26.784,154.884
C05088=1067.273,75.287,429.264,172.625,26.786,154.885
C05089=1067.279,75.537,429.247,172.627,26.789,154.885
C05090=1067.284,75.786,429.229,172.628,26.792,154.885
C05091=1067.290,76.036,429.211,172.630,26.795,154.886
C05092=1067.297,76.284,429.194,172.631,26.797,154.886
C05093=1067.303,76.534,429.176,172.633,26.800,154.886
C05094=1067.308,76.783,429.159,172.634,26.803,154.887
C05095=1067.314,77.033,429.141,172.635,26.806,154.887
C05096=1067.320,77.281,429.122,172.637,26.808,154.888
C05097=1067.326,77.530,429.105,172.638,26.811,154.888
C05098=1067.332,77.780,429.087,172.640,26.814,154.888
C05099=1067.337,78.029,429.069,172.641,26.817,154.889
C05100=1067.345,78.312,429.049,172.644,26.820,154.889
C05101=1067.351,78.596,429.029,172.645,26.823,154.890
C05102=1067.358,78.879,429.009,172.646,26.826,154.890
C05103=1067.364,79.162,428.989,172.648,26.829,154.890
C05104=1067.370,79.412,428.971,172.649,26.832,154.891
C05105=1067.376,79.661,428.953,172.651,26.834,154.891
C05106=1067.382,79.911,428.935,172.652,26.837,154.892
C05107=1067.388,80.159,428.917,172.654,26.840,154.892
C05108=1067.394,80.409,428.899,172.655,26.843,154.892
C05109=1067.399,80.658,428.881,172.657,26.845,154.893
C05110=1067.405,80.907,428.864,172.658,26.848,154.893
C05111=1067.411,81.157,428.846,172.660,26.851,154.893
C05112=1067.417,81.405,428.828,172.661,26.854,154.894
C05113=1067.423,81.655,428.810,172.662,26.856,154.894
C05114=1067.428,81.904,428.791,172.664,26.859,154.895
C05115=1067.434,82.154,428.774,172.665,26.862,154.895
C05116=1067.439,82.403,428.756,172.667,26.864,154.895
C05117=1067.446,82.652,428.737,172.668,26.867,154.896
C05118=1067.452,82.902,428.719,172.670,26.870,154.896
C05119=1067.457,83.151,428.702,172.671,26.873,154.897
C05120=1067.464,83.401,428.684,172.673,26.876,154.897
C05121=1067.469,83.649,428.666,172.674,26.878,154.897
C05122=1067.475,83.899,428.648,172.676,26.881,154.898
C05123=1067.481,84.148,428.630,172.677,26.884,154.898
C05124=1067.487,84.397,428.611,172.679,26.886,154.898
C05125=1067.492,84.646,428.593,172.680,26.889,154.899
C05126=1067.498,84.896,428.575,172.681,26.892,154.899
C05127=1067.504,85.144,428.557,172.683,26.895,154.900
C05128=1067.510,85.394,428.539,172.684,26.897,154.900
C05129=1067.516,85.644,428.521,172.686,26.900,154.900
C05130=1067.522,85.892,428.503,172.687,26.903,154.901
C05131=1067.528,86.142,428.485,172.689,26.906,154.901
C05132=1067.533,86.391,428.467,172.690,26.908,154.902
C05133=1067.540,86.641,428.448,172.692,26.911,154.902
C05134=1067.546,86.890,428.430,172.693,26.913,154.902
C05135=1067.551,87.139,428.413,172.695,26.916,154.903
C05136=1067.558,87.388,428.394,172.696,26.919,154.903
C05137=1067.563,87.637,428.376,172.698,26.922,154.903
C05138=1067.570,87.887,428.358,172.699,26.924,154.904
C05139=1067.575,88.137,428.339,172.701,26.927,154.904
C05140=1067.580,88.386,428.322,172.703,26.930,154.904
C05141=1067.587,88.635,428.303,172.704,26.933,154.905
C05142=1067.593,88.885,428.285,172.706,26.935,154.905
C05143=1067.599,89.133,428.267,172.708,26.938,154.906
C05144=1067.605,89.383,428.249,172.709,26.941,154.906
C05145=1067.610,89.631,428.230,172.710,26.944,154.906
C05146=1067.616,89.881,428.212,172.712,26.946,154.907
C05147=1067.623,90.130,428.193,172.713,26.949,154.907
C05148=1067.628,90.379,428.176,172.715,26.952,154.907
C05149=1067.634,90.628,428.157,172.716,26.954,154.908
C05150=1067.640,90.879,428.139,172.718,26.957,154.908
C05151=1067.646,91.127,428.120,172.719,26.960,154.909
C05152=1067.652,91.377,428.103,172.721,26.962,154.909
C05153=1067.658,91.626,428.083,172.722,26.965,154.909
C05154=1067.663,91.875,428.066,172.724,26.968,154.910
C05155=1067.669,92.124,428.047,172.725,26.971,154.910
C05156=1067.675,92.374,428.029,172.727,26.974,154.911
C05157=1067.681,92.623,428.010,172.728,26.976,154.911
C05158=1067.686,92.872,427.991,172.730,26.979,154.911
C05159=1067.692,93.121,427.973,172.731,26.981,154.912
C05160=1067.698,93.370,427.955,172.733,26.984,154.912
C05161=1067.704,93.620,427.936,172.734,26.987,154.912
C05162=1067.709,93.869,427.918,172.735,26.990,154.913
C05163=1067.715,94.118,427.899,172.737,26.993,154.913
C05164=1067.722,94.402,427.878,172.738,26.996,154.914
C05165=1067.729,94.685,427.857,172.741,26.999,154.914
C05166=1067.735,94.968,427.836,172.742,27.002,154.914
C05167=1067.742,95.251,427.815,172.744,27.005,154.915
C05168=1067.748,95.500,427.796,172.745,27.008,154.915
C05169=1067.753,95.749,427.778,172.747,27.010,154.916
C05170=1067.759,95.999,427.760,172.748,27.013,154.916
C05171=1067.765,96.248,427.740,172.749,27.016,154.917
C05172=1067.771,96.498,427.722,172.751,27.018,154.917
C05173=1067.777,96.747,427.704,172.752,27.021,154.917
C05174=1067.783,96.996,427.685,172.755,27.024,154.918
C05175=1067.789,97.245,427.666,172.756,27.027,154.918
C05176=1067.794,97.494,427.647,172.758,27.030,154.918
C05177=1067.800,97.744,427.629,172.759,27.033,154.919
C05178=1067.806,97.993,427.610,172.761,27.035,154.919
C05179=1067.812,98.242,427.592,172.762,27.038,154.919
C05180=1067.817,98.491,427.573,172.764,27.041,154.920
C05181=1067.824,98.741,427.555,172.765,27.043,154.920
C05182=1067.829,98.990,427.536,172.767,27.046,154.921
C05183=1067.836,99.239,427.517,172.768,27.048,154.921
C05184=1067.842,99.488,427.498,172.770,27.051,154.921
C05185=1067.847,99.737,427.479,172.771,27.054,154.922
C05186=1067.853,99.987,427.461,172.773,27.057,154.922
C05187=1067.859,100.236,427.442,172.774,27.059,154.922
C05188=1067.865,100.485,427.424,172.776,27.062,154.923
C05189=1067.870,100.734,427.405,172.777,27.065,154.923
C05190=1067.877,100.983,427.386,172.779,27.068,154.924
C05191=1067.883,101.233,427.367,172.780,27.070,154.924
C05192=1067.888,101.482,427.347,172.782,27.073,154.924
C05193=1067.895,101.731,427.329,172.783,27.075,154.925
C05194=1067.899,101.980,427.311,172.785,27.078,154.925
C05195=1067.905,102.230,427.291,172.787,27.081,154.925
C05196=1067.912,102.479,427.273,172.788,27.084,154.926
C05197=1067.917,102.728,427.254,172.790,27.087,154.926
C05198=1067.922,102.977,427.235,172.791,27.090,154.927
C05199=1067.929,103.226,427.216,172.793,27.093,154.927
C05200=1067.934,103.476,427.197,172.794,27.095,154.927
C05201=1067.940,103.725,427.178,172.796,27.098,154.928
C05202=1067.947,103.974,427.159,172.797,27.100,154.928
C05203=1067.952,104.223,427.140,172.799,27.103,154.929
C05204=1067.957,104.472,427.121,172.800,27.106,154.929
C05205=1067.963,104.722,427.102,172.802,27.109,154.929
C05206=1067.969,104.971,427.083,172.803,27.112,154.930
C05207=1067.975,105.220,427.064,172.805,27.114,154.930
C05208=1067.980,105.469,427.045,172.806,27.117,154.930
C05209=1067.987,105.718,427.026,172.808,27.120,154.931
C05210=1067.992,105.968,427.007,172.809,27.122,154.931
C05211=1067.998,106.217,426.988,172.812,27.125,154.932
C05212=1068.004,106.467,426.968,172.813,27.128,154.932
C05213=1068.010,106.716,426.950,172.815,27.130,154.932
C05214=1068.015,106.964,426.931,172.816,27.133,154.933
C05215=1068.021,107.214,426.912,172.818,27.136,154.933
C05216=1068.027,107.463,426.892,172.819,27.139,154.934
C05217=1068.033,107.712,426.874,172.821,27.142,154.934
C05218=1068.039,107.961,426.854,172.822,27.144,154.934
C05219=1068.045,108.211,426.835,172.824,27.147,154.935
C05220=1068.051,108.460,426.816,172.825,27.150,154.935
C05221=1068.057,108.709,426.797,172.827,27.152,154.935
C05222=1068.062,108.958,426.778,172.828,27.155,154.936
C05223=1068.068,109.207,426.758,172.830,27.158,154.936
C05224=1068.073,109.457,426.739,172.831,27.160,154.937
C05225=1068.080,109.705,426.720,172.833,27.163,154.937
C05226=1068.086,109.955,426.701,172.835,27.166,154.937
C05227=1068.091,110.204,426.681,172.836,27.169,154.938
C05228=1068.099,110.488,426.660,172.838,27.172,154.938
C05229=1068.105,110.771,426.638,172.839,27.174,154.939
C05230=1068.112,111.054,426.616,172.842,27.178,154.939
C05231=1068.118,111.337,426.594,172.843,27.181,154.939
C05232=1068.124,111.586,426.575,172.845,27.184,154.940
C05233=1068.129,111.836,426.556,172.846,27.186,154.940
C05234=1068.136,112.085,426.537,172.849,27.189,154.940
C05235=1068.142,112.334,426.517,172.850,27.192,154.941
C05236=1068.147,112.583,426.498,172.852,27.195,154.941
C05237=1068.153,112.832,426.478,172.853,27.197,154.942
C05238=1068.159,113.081,426.458,172.855,27.200,154.942
C05239=1068.165,113.331,426.439,172.856,27.202,154.942
C05240=1068.170,113.580,426.420,172.858,27.205,154.943
C05241=1068.176,113.830,426.401,172.859,27.208,154.943
C05242=1068.182,114.078,426.381,172.861,27.211,154.944
C05243=1068.188,114.328,426.362,172.862,27.214,154.944
C05244=1068.193,114.577,426.343,172.864,27.216,154.944
C05245=1068.199,114.825,426.323,172.866,27.220,154.945
C05246=1068.205,115.075,426.303,172.867,27.222,154.945
C05247=1068.211,115.324,426.284,172.869,27.225,154.945
C05248=1068.216,115.573,426.264,172.871,27.227,154.946
C05249=1068.222,115.822,426.245,172.872,27.230,154.946
C05250=1068.228,116.071,426.225,172.873,27.233,154.947
C05251=1068.233,116.321,426.205,172.875,27.236,154.947
C05252=1068.239,116.570,426.185,172.876,27.239,154.947
C05253=1068.245,116.819,426.166,172.878,27.241,154.948
C05254=1068.250,117.069,426.147,172.879,27.244,154.948
C05255=1068.256,117.318,426.127,172.882,27.247,154.949
C05256=1068.262,117.567,426.108,172.883,27.250,154.949
C05257=1068.267,117.815,426.088,172.885,27.253,154.949
C05258=1068.272,118.065,426.068,172.886,27.255,154.950
C05259=1068.278,118.314,426.048,172.888,27.258,154.950
C05260=1068.284,118.563,426.029,172.889,27.261,154.951
C05261=1068.290,118.812,426.009,172.891,27.263,154.951
C05262=1068.296,119.061,425.990,172.892,27.266,154.951
C05263=1068.302,119.310,425.970,172.894,27.269,154.952
C05264=1068.307,119.560,425.950,172.896,27.272,154.952
C05265=1068.313,119.809,425.930,172.898,27.275,154.953
C05266=1068.318,120.058,425.911,172.899,27.277,154.953
C05267=1068.324,120.307,425.891,172.901,27.280,154.953
C05268=1068.330,120.556,425.872,172.902,27.283,154.954
C05269=1068.336,120.805,425.852,172.904,27.286,154.954
C05270=1068.341,121.054,425.831,172.905,27.288,154.954
C05271=1068.347,121.304,425.812,172.907,27.291,154.955
C05272=1068.353,121.553,425.792,172.909,27.294,154.955
C05273=1068.359,121.802,425.773,172.911,27.296,154.956
C05274=1068.365,122.051,425.752,172.912,27.299,154.956
C05275=1068.371,122.300,425.732,172.914,27.302,154.956
C05276=1068.376,122.550,425.712,172.915,27.305,154.957
C05277=1068.382,122.799,425.693,172.917,27.308,154.957
C05278=1068.388,123.048,425.673,172.918,27.310,154.958
C05279=1068.394,123.297,425.653,172.920,27.313,154.958
C05280=1068.400,123.546,425.633,172.922,27.316,154.958
C05281=1068.405,123.796,425.614,172.924,27.318,154.959
C05282=1068.411,124.044,425.594,172.925,27.321,154.959
C05283=1068.417,124.293,425.574,172.927,27.324,154.959
C05284=1068.423,124.542,425.554,172.928,27.327,154.960
C05285=1068.428,124.792,425.534,172.930,27.329,154.960
C05286=1068.434,125.041,425.514,172.931,27.332,154.961
C05287=1068.440,125.290,425.494,172.934,27.335,154.961
C05288=1068.446,125.540,425.474,172.935,27.338,154.961
C05289=1068.452,125.788,425.454,172.937,27.340,154.962
C05290=1068.457,126.038,425.434,172.938,27.343,154.962
C05291=1068.463,126.286,425.414,172.940,27.345,154.962
C05292=1068.470,126.570,425.391,172.942,27.349,154.963
C05293=1068.477,126.853,425.368,172.944,27.352,154.963
C05294=1068.483,127.136,425.345,172.946,27.355,154.964
C05295=1068.489,127.419,425.323,172.947,27.358,154.964
C05296=1068.496,127.668,425.303,172.949,27.361,154.964
C05297=1068.501,127.918,425.283,172.950,27.363,154.965
C05298=1068.507,128.166,425.263,172.953,27.366,154.965
C05299=1068.513,128.416,425.243,172.954,27.369,154.966
C05300=1068.519,128.665,425.223,172.956,27.371,154.966
C05301=1068.525,128.915,425.202,172.957,27.374,154.966
C05302=1068.531,129.163,425.183,172.959,27.377,154.967
C05303=1068.537,129.412,425.163,172.961,27.379,154.967
C05304=1068.543,129.661,425.143,172.963,27.382,154.967
C05305=1068.548,129.910,425.122,172.964,27.385,154.968
C05306=1068.555,130.160,425.102,172.966,27.388,154.968
C05307=1068.560,130.409,425.082,172.968,27.390,154.968
C05308=1068.566,130.658,425.062,172.969,27.393,154.969
C05309=1068.572,130.907,425.042,172.971,27.396,154.969
C05310=1068.578,131.156,425.022,172.973,27.399,154.970
C05311=1068.584,131.405,425.002,172.975,27.401,154.970
C05312=1068.589,131.654,424.981,172.976,27.404,154.970
C05313=1068.595,131.903,424.961,172.978,27.406,154.971
C05314=1068.601,132.152,424.941,172.979,27.409,154.971
C05315=1068.607,132.402,424.920,172.981,27.412,154.972
C05316=1068.616,132.787,424.889,172.984,27.416,154.972
C05317=1068.625,133.174,424.857,172.986,27.421,154.973
C05318=1068.633,133.559,424.826,172.989,27.425,154.973
C05319=1068.643,133.945,424.794,172.992,27.429,154.974
C05320=1068.648,134.194,424.773,172.993,27.431,154.974
C05321=1068.654,134.443,424.753,172.995,27.434,154.975
C05322=1068.659,134.692,424.733,172.997,27.437,154.975
C05323=1068.665,134.942,424.712,172.998,27.440,154.975
C05324=1068.671,135.191,424.692,173.000,27.443,154.976
C05325=1068.676,135.440,424.672,173.002,27.445,154.976
C05326=1068.682,135.689,424.652,173.003,27.448,154.977
C05327=1068.688,135.938,424.631,173.006,27.451,154.977
C05328=1068.694,136.187,424.611,173.007,27.454,154.977
C05329=1068.700,136.436,424.590,173.009,27.456,154.978
C05330=1068.706,136.685,424.569,173.010,27.459,154.978
C05331=1068.712,136.934,424.549,173.012,27.461,154.978
C05332=1068.717,137.184,424.528,173.014,27.465,154.979
C05333=1068.723,137.432,424.508,173.016,27.467,154.979
C05334=1068.729,137.682,424.487,173.017,27.470,154.980
C05335=1068.735,137.931,424.467,173.019,27.473,154.980
C05336=1068.740,138.180,424.446,173.020,27.476,154.980
C05337=1068.746,138.429,424.425,173.023,27.478,154.981
C05338=1068.752,138.678,424.405,173.024,27.481,154.981
C05339=1068.758,138.927,424.384,173.026,27.484,154.981
C05340=1068.763,139.176,424.363,173.027,27.486,154.982
C05341=1068.770,139.425,424.343,173.030,27.490,154.982
C05342=1068.775,139.674,424.322,173.031,27.492,154.983
C05343=1068.780,139.924,424.302,173.033,27.495,154.983
C05344=1068.787,140.172,424.281,173.034,27.497,154.983
C05345=1068.792,140.422,424.260,173.036,27.500,154.984
C05346=1068.798,140.671,424.240,173.038,27.503,154.984
C05347=1068.803,140.920,424.219,173.040,27.506,154.985
C05348=1068.810,141.169,424.198,173.041,27.509,154.985
C05349=1068.815,141.418,424.177,173.043,27.511,154.985
C05350=1068.820,141.667,424.157,173.045,27.514,154.986
C05351=1068.826,141.916,424.135,173.047,27.517,154.986
C05352=1068.836,142.312,424.103,173.049,27.521,154.987
C05353=1068.845,142.707,424.069,173.052,27.526,154.987
C05354=1068.853,143.102,424.037,173.054,27.530,154.988
C05355=1068.862,143.497,424.004,173.058,27.534,154.989
C05356=1068.868,143.746,423.982,173.059,27.537,154.989
C05357=1068.874,143.995,423.962,173.061,27.539,154.989
C05358=1068.880,144.244,423.941,173.063,27.542,154.990
C05359=1068.886,144.494,423.920,173.065,27.545,154.990
C05360=1068.891,144.742,423.899,173.066,27.548,154.990
C05361=1068.897,144.992,423.878,173.068,27.551,154.991
C05362=1068.902,145.241,423.857,173.070,27.554,154.991
C05363=1068.909,145.489,423.837,173.072,27.556,154.991
C05364=1068.915,145.739,423.816,173.073,27.559,154.992
C05365=1068.920,145.988,423.794,173.075,27.562,154.992
C05366=1068.926,146.237,423.773,173.077,27.565,154.993
C05367=1068.932,146.486,423.752,173.079,27.567,154.993
C05368=1068.937,146.735,423.732,173.080,27.570,154.993
C05369=1068.944,146.984,423.711,173.082,27.572,154.994
C05370=1068.949,147.232,423.689,173.084,27.575,154.994
C05371=1068.955,147.482,423.668,173.086,27.578,154.995
C05372=1068.961,147.731,423.647,173.087,27.581,154.995
C05373=1068.967,147.981,423.626,173.090,27.584,154.995
C05374=1068.972,148.229,423.605,173.091,27.587,154.996
C05375=1068.977,148.478,423.584,173.093,27.589,154.996
C05376=1068.984,148.727,423.563,173.094,27.592,154.996
C05377=1068.989,148.976,423.541,173.097,27.595,154.997
C05378=1068.995,149.226,423.521,173.098,27.597,154.997
C05379=1069.001,149.474,423.499,173.100,27.600,154.998
C05380=1069.006,149.724,423.478,173.101,27.603,154.998
C05381=1069.012,149.973,423.457,173.104,27.606,154.998
C05382=1069.018,150.222,423.435,173.105,27.609,154.999
C05383=1069.023,150.471,423.415,173.107,27.611,154.999
C05384=1069.029,150.719,423.394,173.109,27.614,154.999
C05385=1069.035,150.969,423.372,173.111,27.617,155.000
C05386=1069.041,151.217,423.351,173.112,27.620,155.000
C05387=1069.047,151.467,423.330,173.114,27.622,155.001
C05388=1069.052,151.715,423.309,173.116,27.625,155.001
C05389=1069.058,151.965,423.287,173.118,27.628,155.002
C05390=1069.064,152.214,423.266,173.119,27.631,155.002
C05391=1069.070,152.463,423.245,173.122,27.633,155.002
C05392=1069.075,152.711,423.223,173.124,27.636,155.003
C05393=1069.081,152.961,423.201,173.125,27.639,155.003
C05394=1069.086,153.209,423.180,173.127,27.642,155.003
C05395=1069.092,153.459,423.159,173.129,27.645,155.004
C05396=1069.098,153.708,423.138,173.131,27.647,155.004
C05397=1069.104,153.957,423.116,173.132,27.650,155.005
C05398=1069.109,154.206,423.095,173.135,27.653,155.005
C05399=1069.116,154.455,423.073,173.136,27.655,155.005
C05400=1069.121,154.704,423.053,173.138,27.658,155.006
C05401=1069.127,154.953,423.031,173.140,27.661,155.006
C05402=1069.133,155.202,423.010,173.142,27.664,155.006
C05403=1069.138,155.451,422.987,173.143,27.667,155.007
C05404=1069.143,155.700,422.966,173.146,27.670,155.007
C05405=1069.150,155.949,422.945,173.147,27.673,155.008
C05406=1069.155,156.197,422.923,173.149,27.675,155.008
C05407=1069.161,156.447,422.902,173.151,27.678,155.008
C05408=1069.166,156.697,422.880,173.153,27.681,155.009
C05409=1069.172,156.945,422.859,173.154,27.683,155.009
C05410=1069.178,157.194,422.837,173.157,27.686,155.010
C05411=1069.184,157.443,422.816,173.158,27.689,155.010
C05412=1069.189,157.692,422.794,173.160,27.692,155.010
C05413=1069.195,157.941,422.772,173.161,27.695,155.011
C05414=1069.201,158.190,422.751,173.164,27.698,155.011
C05415=1069.207,158.439,422.729,173.165,27.700,155.012
C05416=1069.214,158.722,422.705,173.168,27.703,155.012
C05417=1069.220,159.005,422.681,173.169,27.706,155.012
C05418=1069.226,159.287,422.655,173.172,27.710,155.013
C05419=1069.232,159.570,422.631,173.174,27.713,155.013
C05420=1069.239,159.819,422.609,173.176,27.716,155.014
C05421=1069.244,160.068,422.588,173.177,27.718,155.014
C05422=1069.250,160.317,422.566,173.180,27.721,155.014
C05423=1069.256,160.566,422.544,173.181,27.724,155.015
C05424=1069.261,160.815,422.522,173.184,27.727,155.015
C05425=1069.267,161.064,422.501,173.185,27.729,155.015
C05426=1069.273,161.314,422.479,173.187,27.732,155.016
C05427=1069.278,161.562,422.457,173.189,27.735,155.016
C05428=1069.284,161.812,422.435,173.191,27.738,155.017
C05429=1069.290,162.059,422.413,173.192,27.741,155.017
C05430=1069.295,162.309,422.391,173.195,27.744,155.018
C05431=1069.301,162.557,422.370,173.196,27.747,155.018
C05432=1069.306,162.807,422.347,173.198,27.750,155.018
C05433=1069.311,163.056,422.326,173.200,27.753,155.019
C05434=1069.317,163.305,422.304,173.202,27.755,155.019
C05435=1069.323,163.554,422.281,173.203,27.758,155.020
C05436=1069.328,163.802,422.260,173.206,27.761,155.020
C05437=1069.334,164.052,422.237,173.207,27.764,155.020
C05438=1069.339,164.301,422.216,173.209,27.767,155.021
C05439=1069.345,164.549,422.193,173.211,27.770,155.021
C05440=1069.351,164.799,422.171,173.213,27.772,155.022
C05441=1069.356,165.047,422.150,173.215,27.775,155.022
C05442=1069.361,165.297,422.128,173.217,27.778,155.022
C05443=1069.367,165.545,422.105,173.218,27.781,155.023
C05444=1069.373,165.794,422.083,173.221,27.784,155.023
C05445=1069.378,166.044,422.061,173.222,27.787,155.024
C05446=1069.383,166.292,422.038,173.224,27.790,155.024
C05447=1069.390,166.541,422.017,173.226,27.793,155.024
C05448=1069.395,166.791,421.995,173.228,27.795,155.025
C05449=1069.401,167.039,421.973,173.230,27.798,155.025
C05450=1069.406,167.288,421.950,173.232,27.801,155.026
C05451=1069.412,167.538,421.928,173.233,27.804,155.026
C05452=1069.418,167.785,421.906,173.236,27.807,155.026
C05453=1069.423,168.035,421.884,173.237,27.810,155.027
C05454=1069.428,168.284,421.862,173.240,27.813,155.027
C05455=1069.434,168.532,421.840,173.242,27.815,155.028
C05456=1069.440,168.782,421.818,173.243,27.818,155.028
C05457=1069.445,169.031,421.795,173.246,27.821,155.028
C05458=1069.452,169.280,421.773,173.247,27.824,155.029
C05459=1069.457,169.528,421.750,173.250,27.827,155.029
C05460=1069.462,169.778,421.728,173.251,27.830,155.030
C05461=1069.468,170.027,421.706,173.253,27.832,155.030
C05462=1069.473,170.275,421.684,173.255,27.835,155.030
C05463=1069.479,170.525,421.662,173.257,27.838,155.031
C05464=1069.485,170.773,421.639,173.259,27.841,155.031
C05465=1069.491,171.023,421.617,173.261,27.844,155.032
C05466=1069.496,171.271,421.595,173.263,27.847,155.032
